fbCase_tests(
	bExecute:= TRUE, 
	bDoorReject:= bDoorReject, 
	stDoorGuardReject:= stCaseRejectReasons_tests.stDoorGuardReject, 
	stProductInstruction:= stProductInstruction_tests, 
	stCodeInfo_Outer:= stCodeInfo_Outer_tests, 
	stCACData:= stCACData_tests, 
	stCACDataHMI:= stCACDataHMI_tests, 
	bDone=> bDone, 
	bBusy=> bBusy, 
	bCACValid=> bCACValid, 
	bCACInvalid=> bCACInvalid, 
	bCheckDuplicates=> bCheckDuplicates, 
	bReadyToValidate=> bReadyToValidate, 
	sRejectCode=> sRejectCode_tests, 
	sCaseContent=> sCaseContent_tests);

bEqualCaseBarcodeCheck := (sTempCaseBarcode = stCACDataHMI_tests.sBarcode);

AssertEquals_BOOL(Expected := TRUE,
                  Actual := bEqualCaseBarcodeCheck,
                  Message := 'HMICaseBarcode not OK on valida data'
);

AssertEquals_STRING(Expected := TO_STRING(sTempCaseBarcode),
                    Actual := TO_STRING(stCACDataHMI_tests.sBarcode),
                    Message := 'HMICaseBarcode String Compare FALSE');
						

TEST_FINISHED();
END_METHOD

METHOD INTERNAL dataHMI02_CaseBarcodeOkOnInalidData
VAR
	fbCase_tests		: FB_CASE_FinaliseData;
	
	bDoorReject			: BOOL;	
	bDone 				: BOOL;
	bBusy				: BOOL;

	bCACValid			: BOOL;
	bCACInvalid			: BOOL;

	bCheckDuplicates	: BOOL;
	bReadyToValidate	: BOOL;
	
	sTempCaseBarcode		: T_CASE_Barcode;
	bEqualCaseBarcodeCheck	: BOOL;			
		
END_VAR

//Data initialization
TestInit(stCACData:= stCACData_tests, stProductInstruction:= stProductInstruction_tests);

//Change some data for test scenario below
stCACData_tests.CaseRejectCode := ''; // data not OK
stCACData_tests.Barcode := 'CaseBarcode';
sTempCaseBarcode := F_CONCAT3(stCACData_tests.Barcode,'(999)','0');
	
TcUnit.TEST('dataHMI02_CaseBarcodeOkOnInalidData');

fbCase_tests(
	bExecute:= TRUE, 
	bDoorReject:= bDoorReject, 
	stDoorGuardReject:= stCaseRejectReasons_tests.stDoorGuardReject, 
	stProductInstruction:= stProductInstruction_tests, 
	stCodeInfo_Outer:= stCodeInfo_Outer_tests, 
	stCACData:= stCACData_tests, 
	stCACDataHMI:= stCACDataHMI_tests, 
	bDone=> bDone, 
	bBusy=> bBusy, 
	bCACValid=> bCACValid, 
	bCACInvalid=> bCACInvalid, 
	bCheckDuplicates=> bCheckDuplicates, 
	bReadyToValidate=> bReadyToValidate, 
	sRejectCode=> sRejectCode_tests, 
	sCaseContent=> sCaseContent_tests);

bEqualCaseBarcodeCheck := (sTempCaseBarcode = stCACDataHMI_tests.sBarcode);

AssertEquals_BOOL(Expected := TRUE,
                  Actual := bEqualCaseBarcodeCheck,
                  Message := 'HMICaseBarcode not OK on valida data'
);

AssertEquals_STRING(Expected := TO_STRING(sTempCaseBarcode),
                    Actual := TO_STRING(stCACDataHMI_tests.sBarcode),
                    Message := 'HMICaseBarcode String Compare FALSE');
						

TEST_FINISHED();
END_METHOD

METHOD INTERNAL dataHMI03_OuterBarcodeOkOnInalidData
VAR
	fbCase_tests		: FB_CASE_FinaliseData;
	
	bDoorReject			: BOOL;	
	bDone 				: BOOL;
	bBusy				: BOOL;

	bCACValid			: BOOL;
	bCACInvalid			: BOOL;

	bCheckDuplicates	: BOOL;
	bReadyToValidate	: BOOL;
	
	sTempCaseBarcode		: T_CASE_Barcode;
	bEqualCaseBarcodeCheck	: BOOL;			
		
END_VAR

//Data initialization
TestInit(stCACData:= stCACData_tests, stProductInstruction:= stProductInstruction_tests);

//Change some data for test scenario below
stCACData_tests.Outer[1].OuterRejectCode := ''; // data not OK
stCACData_tests.Outer[1].Barcode := 'OuterBarcode';
sTempCaseBarcode := F_CONCAT3(stCACData_tests.Outer[1].Barcode,'(999)','0');
	
TcUnit.TEST('dataHMI03_OuterBarcodeOkOnInalidData');

fbCase_tests(
	bExecute:= TRUE, 
	bDoorReject:= bDoorReject, 
	stDoorGuardReject:= stCaseRejectReasons_tests.stDoorGuardReject, 
	stProductInstruction:= stProductInstruction_tests, 
	stCodeInfo_Outer:= stCodeInfo_Outer_tests, 
	stCACData:= stCACData_tests, 
	stCACDataHMI:= stCACDataHMI_tests, 
	bDone=> bDone, 
	bBusy=> bBusy, 
	bCACValid=> bCACValid, 
	bCACInvalid=> bCACInvalid, 
	bCheckDuplicates=> bCheckDuplicates, 
	bReadyToValidate=> bReadyToValidate, 
	sRejectCode=> sRejectCode_tests, 
	sCaseContent=> sCaseContent_tests);

bEqualCaseBarcodeCheck := (sTempCaseBarcode = stCACDataHMI_tests.aOuter[1].sBarcode);

AssertEquals_BOOL(Expected := TRUE,
                  Actual := bEqualCaseBarcodeCheck,
                  Message := 'HMIOuterBarcode not OK on valida data'
);

AssertEquals_STRING(Expected := TO_STRING(sTempCaseBarcode),
                    Actual := TO_STRING(stCACDataHMI_tests.aOuter[1].sBarcode),
                    Message := 'HMIOuterBarcode String Compare FALSE');
						

TEST_FINISHED();
END_METHOD

METHOD INTERNAL dataHMI04_OuterBarcodeNotOkOnValidData
VAR
	fbCase_tests		: FB_CASE_FinaliseData;
	
	bDoorReject			: BOOL;	
	bDone 				: BOOL;
	bBusy				: BOOL;

	bCACValid			: BOOL;
	bCACInvalid			: BOOL;

	bCheckDuplicates	: BOOL;
	bReadyToValidate	: BOOL;
	
	sTempCaseBarcode		: T_CASE_Barcode;
	bEqualCaseBarcodeCheck	: BOOL;			
		
END_VAR

//Data initialization
TestInit(stCACData:= stCACData_tests, stProductInstruction:= stProductInstruction_tests);

//Change some data for test scenario below
stCACData_tests.Outer[1].OuterRejectCode := 'OK'; // data OK
stCACData_tests.Outer[1].Barcode := 'OuterBarcode';
sTempCaseBarcode := F_CONCAT3(stCACData_tests.Outer[1].Barcode,'(999)','1');
	
TcUnit.TEST('dataHMI04_OuterBarcodeNotOkOnValidData');

fbCase_tests(
	bExecute:= TRUE, 
	bDoorReject:= bDoorReject, 
	stDoorGuardReject:= stCaseRejectReasons_tests.stDoorGuardReject, 
	stProductInstruction:= stProductInstruction_tests, 
	stCodeInfo_Outer:= stCodeInfo_Outer_tests, 
	stCACData:= stCACData_tests, 
	stCACDataHMI:= stCACDataHMI_tests, 
	bDone=> bDone, 
	bBusy=> bBusy, 
	bCACValid=> bCACValid, 
	bCACInvalid=> bCACInvalid, 
	bCheckDuplicates=> bCheckDuplicates, 
	bReadyToValidate=> bReadyToValidate, 
	sRejectCode=> sRejectCode_tests, 
	sCaseContent=> sCaseContent_tests);

bEqualCaseBarcodeCheck := (sTempCaseBarcode = stCACDataHMI_tests.aOuter[1].sBarcode);

AssertEquals_BOOL(Expected := TRUE,
                  Actual := bEqualCaseBarcodeCheck,
                  Message := 'HMIOuterBarcode not OK on valida data'
);

AssertEquals_STRING(Expected := TO_STRING(sTempCaseBarcode),
                    Actual := TO_STRING(stCACDataHMI_tests.aOuter[1].sBarcode),
                    Message := 'HMIOuterBarcode String Compare FALSE'
);
						

TEST_FINISHED();
END_METHOD

METHOD INTERNAL dataHMI05_PackBarcodeOkOnInvalidData
VAR
	fbCase_tests		: FB_CASE_FinaliseData;
	
	bDoorReject			: BOOL;	
	bDone 				: BOOL;
	bBusy				: BOOL;

	bCACValid			: BOOL;
	bCACInvalid			: BOOL;

	bCheckDuplicates	: BOOL;
	bReadyToValidate	: BOOL;
	
	sTempCaseBarcode		: T_CASE_Barcode;
	bEqualCaseBarcodeCheck	: BOOL;			
		
END_VAR

//Data initialization
TestInit(stCACData:= stCACData_tests, stProductInstruction:= stProductInstruction_tests);

//Change some data for test scenario below
stCACData_tests.Outer[2].PackRejectCode[4] 	:= ''; // data not OK
stCACData_tests.Outer[2].PackCode[4] 		:= 'PackBarcode';
sTempCaseBarcode := F_CONCAT3(stCACData_tests.Outer[2].PackCode[4],'(999)','0');
	
TcUnit.TEST('dataHMI05_PackBarcodeOkOnInvalidData');

fbCase_tests(
	bExecute:= TRUE, 
	bDoorReject:= bDoorReject, 
	stDoorGuardReject:= stCaseRejectReasons_tests.stDoorGuardReject, 
	stProductInstruction:= stProductInstruction_tests, 
	stCodeInfo_Outer:= stCodeInfo_Outer_tests, 
	stCACData:= stCACData_tests, 
	stCACDataHMI:= stCACDataHMI_tests, 
	bDone=> bDone, 
	bBusy=> bBusy, 
	bCACValid=> bCACValid, 
	bCACInvalid=> bCACInvalid, 
	bCheckDuplicates=> bCheckDuplicates, 
	bReadyToValidate=> bReadyToValidate, 
	sRejectCode=> sRejectCode_tests, 
	sCaseContent=> sCaseContent_tests);

bEqualCaseBarcodeCheck := (sTempCaseBarcode = stCACDataHMI_tests.aOuter[2].aPackCode[4]);

AssertEquals_BOOL(Expected := TRUE,
                  Actual := bEqualCaseBarcodeCheck,
                  Message := 'HMIPackBarcode not OK on valida data'
);

AssertEquals_STRING(Expected := TO_STRING(sTempCaseBarcode),
                    Actual := TO_STRING(stCACDataHMI_tests.aOuter[2].aPackCode[4]),
                    Message := 'HMIPackBarcode String Compare FALSE'
);
						

TEST_FINISHED();
END_METHOD

METHOD INTERNAL dataHMI06_PackBarcodeNotOkOnValidData
VAR
	fbCase_tests		: FB_CASE_FinaliseData;
	
	bDoorReject			: BOOL;	
	bDone 				: BOOL;
	bBusy				: BOOL;

	bCACValid			: BOOL;
	bCACInvalid			: BOOL;

	bCheckDuplicates	: BOOL;
	bReadyToValidate	: BOOL;
	
	sTempCaseBarcode		: T_CASE_Barcode;
	bEqualCaseBarcodeCheck	: BOOL;			
		
END_VAR

//Data initialization
TestInit(stCACData:= stCACData_tests, stProductInstruction:= stProductInstruction_tests);

//Change some data for test scenario below
stCACData_tests.Outer[4].PackRejectCode[10] 	:= 'OK'; // data not OK
stCACData_tests.Outer[4].PackCode[10] 			:= 'PackBarcode';

sTempCaseBarcode := F_CONCAT3(stCACData_tests.Outer[4].PackCode[10],'(999)','1');
	
TcUnit.TEST('dataHMI06_PackBarcodeNotOkOnValidData');

fbCase_tests(
	bExecute:= TRUE, 
	bDoorReject:= bDoorReject, 
	stDoorGuardReject:= stCaseRejectReasons_tests.stDoorGuardReject, 
	stProductInstruction:= stProductInstruction_tests, 
	stCodeInfo_Outer:= stCodeInfo_Outer_tests, 
	stCACData:= stCACData_tests, 
	stCACDataHMI:= stCACDataHMI_tests, 
	bDone=> bDone, 
	bBusy=> bBusy, 
	bCACValid=> bCACValid, 
	bCACInvalid=> bCACInvalid, 
	bCheckDuplicates=> bCheckDuplicates, 
	bReadyToValidate=> bReadyToValidate, 
	sRejectCode=> sRejectCode_tests, 
	sCaseContent=> sCaseContent_tests);

bEqualCaseBarcodeCheck := (sTempCaseBarcode = stCACDataHMI_tests.aOuter[4].aPackCode[10]);

AssertEquals_BOOL(Expected := TRUE,
                  Actual := bEqualCaseBarcodeCheck,
                  Message := 'HMIPackBarcode not OK on valida data'
);

AssertEquals_STRING(Expected := TO_STRING(sTempCaseBarcode),
                    Actual := TO_STRING(stCACDataHMI_tests.aOuter[4].aPackCode[10]),
                    Message := 'HMIPackBarcode String Compare FALSE'
);
						

TEST_FINISHED();
END_METHOD

METHOD INTERNAL main01_FBExecuted_bDoneTRUE
VAR
	fbCase_tests		: FB_CASE_FinaliseData;
	
	bDoorReject			: BOOL;	
	bDone 				: BOOL;
	bBusy				: BOOL;

	bCACValid			: BOOL;
	bCACInvalid			: BOOL;

	bCheckDuplicates	: BOOL;
	bReadyToValidate	: BOOL;
		
END_VAR

//Data initialization
TestInit(stCACData:= stCACData_tests, stProductInstruction:= stProductInstruction_tests);

//Change some data for test scenario below


	
TcUnit.TEST('main01_FBExecuted_bDoneTRUE');

fbCase_tests(
	bExecute:= TRUE, 
	bDoorReject:= bDoorReject, 
	stDoorGuardReject:= stCaseRejectReasons_tests.stDoorGuardReject, 
	stProductInstruction:= stProductInstruction_tests, 
	stCodeInfo_Outer:= stCodeInfo_Outer_tests, 
	stCACData:= stCACData_tests, 
	stCACDataHMI:= stCACDataHMI_tests, 
	bDone=> bDone, 
	bBusy=> bBusy, 
	bCACValid=> bCACValid, 
	bCACInvalid=> bCACInvalid, 
	bCheckDuplicates=> bCheckDuplicates, 
	bReadyToValidate=> bReadyToValidate, 
	sRejectCode=> sRejectCode_tests, 
	sCaseContent=> sCaseContent_tests);



	
AssertEquals_BOOL( Expected	:= TRUE,
			 	   Actual	:= bDone, 
			 	   Message	:= 'FB_CASE_FinaliseData not executed');
						

TEST_FINISHED();
END_METHOD

METHOD INTERNAL main02_bCACValidTrueOnValidData
VAR
	fbCase_tests		: FB_CASE_FinaliseData;
	
	bDoorReject			: BOOL;	
	bDone 				: BOOL;
	bBusy				: BOOL;

	bCACValid			: BOOL;
	bCACInvalid			: BOOL;

	bCheckDuplicates	: BOOL;
	bReadyToValidate	: BOOL;
		
END_VAR

//Data initialization
TestInit(stCACData:= stCACData_tests, stProductInstruction:= stProductInstruction_tests);

//Change some data for test scenario below


	
TcUnit.TEST('main02_bCACValidTrueOnValidData');

fbCase_tests(
	bExecute:= TRUE, 
	bDoorReject:= bDoorReject, 
	stDoorGuardReject:= stCaseRejectReasons_tests.stDoorGuardReject, 
	stProductInstruction:= stProductInstruction_tests, 
	stCodeInfo_Outer:= stCodeInfo_Outer_tests, 
	stCACData:= stCACData_tests, 
	stCACDataHMI:= stCACDataHMI_tests, 
	bDone=> bDone, 
	bBusy=> bBusy, 
	bCACValid=> bCACValid, 
	bCACInvalid=> bCACInvalid, 
	bCheckDuplicates=> bCheckDuplicates, 
	bReadyToValidate=> bReadyToValidate, 
	sRejectCode=> sRejectCode_tests, 
	sCaseContent=> sCaseContent_tests);



	
AssertEquals_BOOL( Expected	:= TRUE,
			 	   Actual	:= bCACValid, 
			 	   Message	:= 'bCACValid wrong value');
						

TEST_FINISHED();
END_METHOD

METHOD INTERNAL main03_bCACInvalidFalseOnValidData
VAR
	fbCase_tests		: FB_CASE_FinaliseData;
	
	bDoorReject			: BOOL;	
	bDone 				: BOOL;
	bBusy				: BOOL;

	bCACValid			: BOOL;
	bCACInvalid			: BOOL;

	bCheckDuplicates	: BOOL;
	bReadyToValidate	: BOOL;
		
END_VAR

//Data initialization
TestInit(stCACData:= stCACData_tests, stProductInstruction:= stProductInstruction_tests);

//Change some data for test scenario below


	
TcUnit.TEST('main03_bCACInvalidFalseOnValidData');

fbCase_tests(
	bExecute:= TRUE, 
	bDoorReject:= bDoorReject, 
	stDoorGuardReject:= stCaseRejectReasons_tests.stDoorGuardReject, 
	stProductInstruction:= stProductInstruction_tests, 
	stCodeInfo_Outer:= stCodeInfo_Outer_tests, 
	stCACData:= stCACData_tests, 
	stCACDataHMI:= stCACDataHMI_tests, 
	bDone=> bDone, 
	bBusy=> bBusy, 
	bCACValid=> bCACValid, 
	bCACInvalid=> bCACInvalid, 
	bCheckDuplicates=> bCheckDuplicates, 
	bReadyToValidate=> bReadyToValidate, 
	sRejectCode=> sRejectCode_tests, 
	sCaseContent=> sCaseContent_tests);



	
AssertEquals_BOOL( Expected	:= FALSE,
			 	   Actual	:= bCACInvalid, 
			 	   Message	:= 'bCACInvalid wrong value');
						

TEST_FINISHED();
END_METHOD

METHOD INTERNAL main04_bCACInvalidTrueOnInvalidData
VAR
	fbCase_tests		: FB_CASE_FinaliseData;
	
	bDoorReject			: BOOL;	
	bDone 				: BOOL;
	bBusy				: BOOL;

	bCACValid			: BOOL;
	bCACInvalid			: BOOL;

	bCheckDuplicates	: BOOL;
	bReadyToValidate	: BOOL;
		
END_VAR

//Data initialization
TestInit(stCACData:= stCACData_tests, stProductInstruction:= stProductInstruction_tests);

//Change some data for test scenario below
stCACData_tests.CaseRejectCode := '';

	
TcUnit.TEST('main04_bCACInvalidTrueOnInvalidData');

fbCase_tests(
	bExecute:= TRUE, 
	bDoorReject:= bDoorReject, 
	stDoorGuardReject:= stCaseRejectReasons_tests.stDoorGuardReject, 
	stProductInstruction:= stProductInstruction_tests, 
	stCodeInfo_Outer:= stCodeInfo_Outer_tests, 
	stCACData:= stCACData_tests, 
	stCACDataHMI:= stCACDataHMI_tests, 
	bDone=> bDone, 
	bBusy=> bBusy, 
	bCACValid=> bCACValid, 
	bCACInvalid=> bCACInvalid, 
	bCheckDuplicates=> bCheckDuplicates, 
	bReadyToValidate=> bReadyToValidate, 
	sRejectCode=> sRejectCode_tests, 
	sCaseContent=> sCaseContent_tests);



	
AssertEquals_BOOL( Expected	:= TRUE,
			 	   Actual	:= bCACInvalid, 
			 	   Message	:= 'bCACInvalid wrong value');
						

TEST_FINISHED();
END_METHOD

METHOD INTERNAL main05_bCACValidFalseOnInvalidData
VAR
	fbCase_tests		: FB_CASE_FinaliseData;
	
	bDoorReject			: BOOL;	
	bDone 				: BOOL;
	bBusy				: BOOL;

	bCACValid			: BOOL;
	bCACInvalid			: BOOL;

	bCheckDuplicates	: BOOL;
	bReadyToValidate	: BOOL;
		
END_VAR

//Data initialization
TestInit(stCACData:= stCACData_tests, stProductInstruction:= stProductInstruction_tests);

//Change some data for test scenario below
stCACData_tests.CaseRejectCode := '';

	
TcUnit.TEST('main05_bCACValidFalseOnInvalidData');

fbCase_tests(
	bExecute:= TRUE, 
	bDoorReject:= bDoorReject, 
	stDoorGuardReject:= stCaseRejectReasons_tests.stDoorGuardReject, 
	stProductInstruction:= stProductInstruction_tests, 
	stCodeInfo_Outer:= stCodeInfo_Outer_tests, 
	stCACData:= stCACData_tests, 
	stCACDataHMI:= stCACDataHMI_tests, 
	bDone=> bDone, 
	bBusy=> bBusy, 
	bCACValid=> bCACValid, 
	bCACInvalid=> bCACInvalid, 
	bCheckDuplicates=> bCheckDuplicates, 
	bReadyToValidate=> bReadyToValidate, 
	sRejectCode=> sRejectCode_tests, 
	sCaseContent=> sCaseContent_tests);



	
AssertEquals_BOOL( Expected	:= FALSE,
			 	   Actual	:= bCACValid, 
			 	   Message	:= 'bCACInvalid wrong value');
						

TEST_FINISHED();
END_METHOD

METHOD INTERNAL main06_FBnotExecuted_bDoneFALSE
VAR
	fbCase_tests		: FB_CASE_FinaliseData;
	
	bDoorReject			: BOOL;	
	bDone 				: BOOL;
	bBusy				: BOOL;

	bCACValid			: BOOL;
	bCACInvalid			: BOOL;

	bCheckDuplicates	: BOOL;
	bReadyToValidate	: BOOL;
		
END_VAR

//Data initialization
TestInit(stCACData:= stCACData_tests, stProductInstruction:= stProductInstruction_tests);

//Change some data for test scenario below


	
TcUnit.TEST('main06_FBnotExecuted_bDoneFALSE');

fbCase_tests(
	bExecute:= FALSE, 
	bDoorReject:= bDoorReject, 
	stDoorGuardReject:= stCaseRejectReasons_tests.stDoorGuardReject, 
	stProductInstruction:= stProductInstruction_tests, 
	stCodeInfo_Outer:= stCodeInfo_Outer_tests, 
	stCACData:= stCACData_tests, 
	stCACDataHMI:= stCACDataHMI_tests, 
	bDone=> bDone, 
	bBusy=> bBusy, 
	bCACValid=> bCACValid, 
	bCACInvalid=> bCACInvalid, 
	bCheckDuplicates=> bCheckDuplicates, 
	bReadyToValidate=> bReadyToValidate, 
	sRejectCode=> sRejectCode_tests, 
	sCaseContent=> sCaseContent_tests);



	
AssertEquals_BOOL( Expected	:= FALSE,
			 	   Actual	:= bDone, 
			 	   Message	:= 'FB_CASE_FinaliseData not executed false');
						

TEST_FINISHED();
END_METHOD

METHOD PUBLIC main07_FBExecuted_bReadyToValidateFALSE
VAR
	fbCase_tests		: FB_CASE_FinaliseData;
	
	bDoorReject			: BOOL;	
	bDone 				: BOOL;
	bBusy				: BOOL;

	bCACValid			: BOOL;
	bCACInvalid			: BOOL;

	bCheckDuplicates	: BOOL;
	bReadyToValidate	: BOOL;
	
		
END_VAR

//Data initialization
TestInit(stCACData:= stCACData_tests, stProductInstruction:= stProductInstruction_tests);

//Change some data for test scenario below


	
TcUnit.TEST('main07_FBExecuted_bReadyToValidateFALSE');

fbCase_tests(
	bExecute:= TRUE, 
	bDoorReject:= bDoorReject, 
	stDoorGuardReject:= stCaseRejectReasons_tests.stDoorGuardReject, 
	stProductInstruction:= stProductInstruction_tests, 
	stCodeInfo_Outer:= stCodeInfo_Outer_tests, 
	stCACData:= stCACData_tests, 
	stCACDataHMI:= stCACDataHMI_tests, 
	bDone=> bDone, 
	bBusy=> bBusy, 
	bCACValid=> bCACValid, 
	bCACInvalid=> bCACInvalid, 
	bCheckDuplicates=> bCheckDuplicates, 
	bReadyToValidate=> bReadyToValidate, 
	sRejectCode=> sRejectCode_tests, 
	sCaseContent=> sCaseContent_tests);



	
AssertEquals_BOOL( Expected	:= TRUE,
			 	   Actual	:= bReadyToValidate, 
			 	   Message	:= 'FB_CASE_FinaliseData executed with bReaduToValidate FALSE');
						

TEST_FINISHED();
END_METHOD

METHOD INTERNAL main08_FBExecuted_bCheckDuplicatesFALSEonOuterDuplicates
VAR
	fbCase_tests		: FB_CASE_FinaliseData;
	
	bDoorReject			: BOOL;	
	bDone 				: BOOL;
	bBusy				: BOOL;

	bCACValid			: BOOL;
	bCACInvalid			: BOOL;

	bCheckDuplicates	: BOOL;
	bReadyToValidate	: BOOL;
		
END_VAR

//Data initialization
TestInit(stCACData:= stCACData_tests, stProductInstruction:= stProductInstruction_tests);

//Change some data for test scenario below
stCACData_tests.Outer[3].Barcode := stCACData_tests.Outer[6].Barcode;

	
TcUnit.TEST('main08_FBExecuted_bCheckDuplicatesFALSEonOuterDuplicates');

fbCase_tests(
	bExecute:= TRUE, 
	bDoorReject:= bDoorReject, 
	stDoorGuardReject:= stCaseRejectReasons_tests.stDoorGuardReject, 
	stProductInstruction:= stProductInstruction_tests, 
	stCodeInfo_Outer:= stCodeInfo_Outer_tests, 
	stCACData:= stCACData_tests, 
	stCACDataHMI:= stCACDataHMI_tests, 
	bDone=> bDone, 
	bBusy=> bBusy, 
	bCACValid=> bCACValid, 
	bCACInvalid=> bCACInvalid, 
	bCheckDuplicates=> bCheckDuplicates, 
	bReadyToValidate=> bReadyToValidate, 
	sRejectCode=> sRejectCode_tests, 
	sCaseContent=> sCaseContent_tests);



	
AssertEquals_BOOL( Expected	:= TRUE,
			 	   Actual	:= bCheckDuplicates, 
			 	   Message	:= 'FB_CASE_FinaliseData executed with bCheckDuplicates FALSE on outer barcode duplicate');
						

TEST_FINISHED();
END_METHOD

METHOD PRIVATE TestInit
VAR_IN_OUT
	stProductInstruction	: ST_PCM_Status;
	stCACData 				: ST_CAC_Data;
END_VAR

VAR	
	rTrigDataInit		: R_TRIG;
	bDataInit			: BOOL;
	iOuter				: INT;
	iPack				: INT;
	sPackNum			: STRING;
	sOuterNum			: STRING;
	sPackCode			: STRING;
END_VAR
	
//MEMSET(ADR(stCACData), 16#00, SIZEOF(stCACData));	

FOR iOuter := 1 TO stProductInstruction.nOutersPerCase DO
	(* Outer number z zerami *)
	sOuterNum := F_StringAddPrefix(INT_TO_STRING(iOuter),2,'0');
	
	(* Write Outers barcodes *)
	stCACData.Outer[iOuter].Barcode    := CONCAT('OUTER', sOuterNum);
	stCACData.Outer[iOuter].OuterCodeStatus := 5;
	stCACData.Outer[iOuter].OuterRejectCode := 'OK';
	
	FOR iPack := 1 TO stProductInstruction.nPacksPerOuter DO
		(* Pack number dwucyfrowy z zerami *)
		sPackNum := F_StringAddPrefix(INT_TO_STRING(iPack),2,'0');			
		(* Sklej pack code *)
		sPackCode := CONCAT(CONCAT('PACK', sPackNum), CONCAT('OUTER', sOuterNum));
		
		(* Write Pack Barcodes / Data*)
		stCACData.Outer[iOuter].PackCode[iPack]			:= sPackCode;
		stCACData.Outer[iOuter].PackCodeStatus[iPack]	:= 5;
		stCACData.Outer[iOuter].PackRejectID[iPack]		:= 0;			
		stCACData.Outer[iOuter].PackRejectCode[iPack]	:= 'OK';
		
					
		stCACData.Outer[iOuter].NumberOfPacks := stProductInstruction.nPacksPerOuter;
		
	END_FOR;
END_FOR;
END_METHOD

END_FUNCTION_BLOCK

// ---- POUs/TcUnit/FB_CASE_DuplicateUpdateToDBTests/FB_CASE_DuplicateUpdateToDBTests.TcPOU
FUNCTION_BLOCK FB_CASE_DuplicateUpdateToDBTests EXTENDS TcUnit.FB_TestSuite

VAR
	
	(* In/Out test 01*)		
	stCACData_01 							: ST_CAC_Data;
	
	stProductInstruction_01		: ST_PCM_Status;
	aOCVPackStatus_01			: ARRAY[1..cMAX_OUTER_STATUS_QUEUE] OF ST_OUTER_Status;	(* Outer status array *)
	aOuterStatus_01				: ARRAY[1..cMAX_OUTER_STATUS_QUEUE] OF ST_OUTER_Status;	(* Outer status array *)
	
	stOCVDataDB_01							: ST_DB_OCVDataCtrl;
	stOACDataDB_01							: ST_DB_OACDataCtrl;
	
	stOuterBarcodeDuplicate_01				: ST_RejectItems;
	stOuterDuplicatedPackCodesFound_01		: ST_RejectItems;
	
	stCodeInfo_Pack_01					: ST_CodeInfo;
	stCodeInfo_Intermediate_01			: ST_CodeInfo;
	stCodeInfo_Outer_01					: ST_CodeInfo;
	
END_VAR

//==============================================================
//MAIN TESTS
//==============================================================

main01_();

METHOD INTERNAL main01_
VAR
	fbCase					: FB_CASE_DuplicateUpdateToDB;
	bIsDuplicateOuter		: BOOL;
	bIsDuplicatePacks		: BOOL;
	

	
END_VAR

//Data initialization
TestInit(stCACData:= stCACData_01, stProductInstruction:= stProductInstruction_01);

//Change some data for test scenario below

	
TcUnit.TEST('main01_');

fbCase(
	bExecute:= TRUE, 
	bUseInterimCodeForValidation:= , 
	aOCVPackStatus:= aOCVPackStatus_01, 
	aOuterStatus:= aOCVPackStatus_01, 
	stOCVDataDB:= stOCVDataDB_01, 
	stOACDataDB:= stOACDataDB_01, 
	stOuterBarcodeDuplicate:=  stOuterBarcodeDuplicate_01, 
	stOuterDuplicatedPackCodesFound:= stOuterDuplicatedPackCodesFound_01, 
	stCodeInfo_Pack:= stCodeInfo_Pack_01, 
	stCodeInfo_Intermediate:= stCodeInfo_Intermediate_01, 
	stCodeInfo_Outer:= stCodeInfo_Outer_01, 
	stCACData:= stCACData_01, 
	bDone=> , 
	bBusy=> , 
	bError=> , 
	nErrorID=> , 
	nOACFilesBlocked=> , 
	nOCVFilesBlocked=> , 
	stDaigOACDataDB=> , 
	stDiagOCVDataDB=> );

	
// AssertEquals_BOOL( Expected	:= ,
// 			 	   Actual	:= , 
// 			 	   Message	:= '');
// 						

TEST_FINISHED();
END_METHOD

METHOD PRIVATE TestInit
VAR_IN_OUT
	stProductInstruction	: ST_PCM_Status;
	stCACData 				: ST_CAC_Data;
END_VAR

VAR	
	rTrigDataInit		: R_TRIG;
	bDataInit			: BOOL;
	iOuter				: INT;
	iPack				: INT;
	sPackNum			: STRING;
	sOuterNum			: STRING;
	sPackCode			: STRING;
END_VAR

stProductInstruction.nOutersPerCase		:= 50;
stProductInstruction.nPacksPerOuter 	:= 10;

stCACData.NumberOfOuters	:= 50;


FOR iOuter := 1 TO stProductInstruction.nOutersPerCase DO
	(* Ustaw outer *)
	stCACData.Outer[iOuter].Barcode    := CONCAT('OUTER', INT_TO_STRING(iOuter));
	stCACData.Outer[iOuter].OuterCodeStatus := 5;
	
	stCACData.Outer[iOuter].OuterRejectID	:= 0;
	
	
	FOR iPack := 1 TO stProductInstruction.nPacksPerOuter DO
		(* Pack number z zerami *)
		sPackNum := CONCAT('0', INT_TO_STRING(iPack));  (* dla 1-9: '01'-'09' *)
		IF iPack = 10 THEN
			sPackNum := '10';
		END_IF;
		
		(* Outer number z zerami dla 1-9 *)
		sOuterNum := CONCAT('0', INT_TO_STRING(iOuter));
		IF iOuter >= 10 THEN
			sOuterNum := INT_TO_STRING(iOuter);
		END_IF;
		
		(* Sklej pack code *)
		sPackCode := CONCAT(CONCAT('PACK', sPackNum), CONCAT('OUTER', sOuterNum));
		
		(* Przypisz *)
		stCACData.Outer[iOuter].PackCode[iPack]			:= sPackCode;
		stCACData.Outer[iOuter].PackCodeStatus[iPack]	:= 5;
		stCACData.Outer[iOuter].PackRejectID[iPack]		:= 0;
		
	END_FOR;
END_FOR;
END_METHOD

END_FUNCTION_BLOCK

// ---- POUs/TcUnit/F_CODE_GetItemAITests/PRG_CODE_GetItemAIManual.TcPOU
PROGRAM PRG_CODE_GetItemAIManual
VAR
	fbCase_DuplicatCheck		: FB_CASE_DuplicatCheck;
	
	(* Init function/method declarations*)
	rTrigDataInit		: R_TRIG;
	bDataInit			: BOOL;
	iOuter				: INT;
	iPack				: INT;
	sPackNum			: STRING;
	sOuterNum			: STRING;
	sPackCode			: STRING;
	
	(* Inputs *)
	bExecute							: BOOL;
	
	(* In/Out *)
	stProductInstruction				: ST_PCM_Status;
	stOuterBarcodeDuplicate				: ST_RejectItems;
	stOuterDuplicatedPackCodesFound		: ST_RejectItems;
	stCaseRejectReasons					: ST_RejectReasonsForCase;
	stRejectReasonForOuters				: ST_RejectReasonsForOuter;	
	stRejectReasonForPacks				: ST_RejectReasonsForPack;	
	
	stCACData 							: ST_CAC_Data;
	
	(* Outputs *)	
	bDone 					: BOOL;
	bBusy					: BOOL;

	bCACValid				: BOOL;
	sRejectCode				: T_MaxString;
	bIsDuplicateOuters		: BOOL;
	bIsDuplicatePacks		: BOOL;
	bReadyToValidate		: BOOL;
	
	stUpdateCACData 		: ST_CAC_Data;
	
	
END_VAR

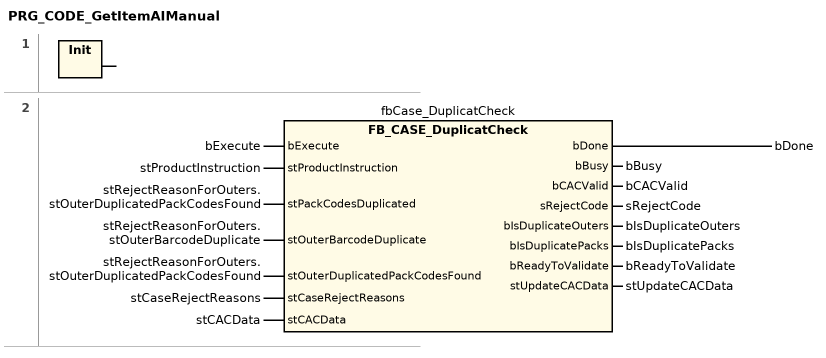
// NETWORK 1
Init();

// NETWORK 2
fbCase_DuplicatCheck(
    bExecute := bExecute,
    stProductInstruction := stProductInstruction,
    stPackCodesDuplicated := stRejectReasonForOuters.stOuterDuplicatedPackCodesFound,
    stOuterBarcodeDuplicate := stRejectReasonForOuters.stOuterBarcodeDuplicate,
    stOuterDuplicatedPackCodesFound := stRejectReasonForOuters.stOuterDuplicatedPackCodesFound,
    stCaseRejectReasons := stCaseRejectReasons,
    stCACData := stCACData,
    bBusy => bBusy,
    bCACValid => bCACValid,
    sRejectCode => sRejectCode,
    bIsDuplicateOuters => bIsDuplicateOuters,
    bIsDuplicatePacks => bIsDuplicatePacks,
    bReadyToValidate => bReadyToValidate,
    stUpdateCACData => stUpdateCACData); // FB_CASE_DuplicatCheck
bDone := fbCase_DuplicatCheck.bDone;

ACTION Init:

rTrigDataInit(CLK := bDataInit);

IF rTrigDataInit.Q THEN
	
stProductInstruction.nOutersPerCase		:= 50;
stProductInstruction.nPacksPerOuter 	:= 10;

	FOR iOuter := 1 TO stProductInstruction.nOutersPerCase DO
		(* Outer number z zerami *)
		sOuterNum := F_StringAddPrefix(INT_TO_STRING(iOuter),2,'0');
		
		(* Write Outers barcodes *)
		stCACData.Outer[iOuter].Barcode    := CONCAT('OUTER', sOuterNum);
		stCACData.Outer[iOuter].OuterCodeStatus := 5;
		
		FOR iPack := 1 TO stProductInstruction.nPacksPerOuter DO
			(* Pack number dwucyfrowy z zerami *)
			sPackNum := F_StringAddPrefix(INT_TO_STRING(iPack),2,'0');			
			(* Sklej pack code *)
			sPackCode := CONCAT(CONCAT('PACK', sPackNum), CONCAT('OUTER', sOuterNum));
			
			(* Write Pack Barcodes *)
			stCACData.Outer[iOuter].PackCode[iPack]			:= sPackCode;
			stCACData.Outer[iOuter].PackCodeStatus[iPack]	:= 5;
			stCACData.Outer[iOuter].PackRejectID[iPack]		:= 0;
			
		END_FOR;
	END_FOR;	
	
END_IF
END_ACTION

END_PROGRAM

// ---- POUs/_Utilites/Addtionals/FB_PulseGenerator_Sync.TcPOU
(* generates one-shot pulses with user-defined period and and sync offset time *)
(* uses GETCPUCOUNTER to synchronise rising edge of timer across multiple FBs *)
FUNCTION_BLOCK FB_PulseGenerator_Sync
VAR_INPUT
	bEnable			: BOOL;		(* set TRUE to enable pulse generation *)
	tPeriod			: TIME;		(* base period for pulse output *)
	nSyncOffset		: DINT;		(* sync offset in ms for rising edge, >0 = phase delay, <0 = phase advance *)
END_VAR
VAR_OUTPUT
	bOutput			: BOOL;		(* one-shot pulse output *)
END_VAR
VAR
	fbCPUCounter	: GETCPUCOUNTER;
	nSystemTime64	: T_ULARGE_INTEGER;
	nSystemTime		: UDINT;
	nLastSystemTime	: UDINT;
END_VAR
(*
-------------------------------------------------------------------------------------------------
Date		Version	Author	Comments
-------------------------------------------------------------------------------------------------
30/01/2015	3.00.00	PB		Initial release

-------------------------------------------------------------------------------------------------
*)

(* enabled and tBaseTime is specified *)
IF bEnable = TRUE AND tPeriod > T#0ms THEN

	(* load global CPU counter value into 64-bit nSystemTime *)
	fbCPUCounter(
		cpuCntLoDW	=> nSystemTime64.dwLowPart,
		cpuCntHiDW	=> nSystemTime64.dwHighPart
	);

	(* phase delay *)
	IF nSyncOffset > 0 THEN

		(* subtract nTimeOffset from system timer *)
		nSystemTime64 := UInt64Sub64(nSystemTime64, UInt32x32To64(ABS(nSyncOffset), 10000));

	(* phase advance *)
	ELSIF nSyncOffset < 0 THEN

		(* add nTimeOffset from system timer *)
		nSystemTime64 := UInt64Add64(nSystemTime64, UInt32x32To64(ABS(nSyncOffset), 10000));
	END_IF

	(* convert nSystemTime from 1= 100ns to 1 = 1ms *)
	nSystemTime64 := UInt64Div64(nSystemTime64, UInt32x32To64(10000, 1));

	(* nSystemTime is sawtooth wave from 0 to tPeriod in ms *)
	nSystemTime := nSystemTime64.dwLowPart MOD TIME_TO_UDINT(tPeriod);

	(* nSystemTime has re-started, convert nLastSystemTime to tPeriod *)
	IF nSystemTime < nLastSystemTime MOD TIME_TO_UDINT(tPeriod) THEN

		bOutput := TRUE;

	(* nSystemTime >= nLastSystemTime *)
	ELSE

		bOutput := FALSE;
	END_IF

	(* store last system time *)
	nLastSystemTime := nSystemTime;

(* disabled or tBaseTime = 0ms *)
ELSE

	bOutput := FALSE;
END_IF

END_FUNCTION_BLOCK

// ---- POUs/_Utilites/Addtionals/PRG_ButtonsHandler.TcPOU
PROGRAM PRG_ButtonsHandler
VAR
	rTrig			: R_TRIG;
	tTimer			: TOF;
	tTriggerTime	: TIME := T#100MS;
	bTimerOn		: BOOL;
END_VAR


rTrig(CLK:= GVL.bSiemensTriggerButton);

tTimer(IN:= bTimerOn, PT:= tTriggerTime);

IF rTrig.Q THEN
	bTimerOn := TRUE;	
ELSIF tTimer.ET = T#0S THEN
	bTimerOn := FALSE;
END_IF

GVL.bSiemensTriggerOutput := tTimer.Q;

END_PROGRAM

// ---- POUs/_Utilites/CAMERAS/FB_SCANNER_HikrobotEXT.TcPOU
FUNCTION_BLOCK FB_SCANNER_HikrobotEXT
VAR_INPUT
	bEnableReceive					: BOOL;
	bEnableSend						: BOOL;
	strScannerIPAddr				: T_IPv4Addr	:= '192.168.1.45';
	nReceiveScannerPortNo			: UINT			:= 2010;
	nSendScannerPortNo				: UINT			:= 4001;	
	stRequestCommand				: E_TCPIP_RequescCommand; (* tutaj powinna byc strukruta z eRequestCommand plus parametry: 0,1 etc *)
	bSendCommand					: BOOL;
	bExecutedCommandSend			: BOOL;
END_VAR

VAR_OUTPUT
	eSocketReceiveState		: E_SocketConnectionState;
	eSocketSendState		: E_SocketConnectionState;
END_VAR

VAR
	fbTCPPortCtrl_Receive	: FB_TCP_ClientPortCtrl;
	bReceiveConnected		: BOOL;
	fbTCPortCtrl_Send		: FB_TCP_ClientPortCtrl;
	bSendConnected			: BOOL;
	fbTCPReceive			: FB_ReceiveString;
	bReceiveExpected		: BOOL;
	fbTCPReceiveAfterSend	: FB_ReceiveString;	
	strTCPRxStringReply		: T_MaxString;
	strTCPRxString			: T_MaxString;
	strTCPRxString_Reply	: T_MaxString;
	ftrigEnable				: F_TRIG;
	bReInitialiseTCP		: BOOL;
	fbTON_TcpTimeout		: TON;
	
	nIndex					: UINT;
	nIndexReply				: UINT;
	nIndex2					: UINT;
	
	/////// send command
	
	fbTCPSend				: FB_SocketSend;
	rTrigSend				: R_TRIG;
	rTrigDataReceived		: R_TRIG;
	rTrigSendCommand		: R_TRIG;
	nCommandNo				: UINT := 1;
	fTrigTCPSendDone		: F_TRIG;
	nSendErrId				: UDINT;
	strTCPCommand			: STRING(20);
	strReplyString			: STRING(20);
	strTCPLastCommand		: STRING(20);
	strLastReplyString		: STRING(20);
	bReplyOK				: BOOL;
	tHeartbeatInterval		: TIME := T#5S;
	eRequestCommand			: E_TCPIP_RequescCommand;
	
	(* SEND SEQUENCE VARIABLE *)
	
	eSendSequenceSTATE		: E_TCPIP_SEND_STATE;
	bSendRequest			: BOOL;
	rTrigSendRequest		: R_TRIG;
END_VAR


Connect();

Receive();

//Send();

Send_Sequence();

ACTION Connect:

(* TCP Receive Socket establish connect *)
fbTCPPortCtrl_Receive(
	bEnable				:= bEnableReceive, 
	strRemoteIPAddr		:= strScannerIPAddr, 
	nRemotePortNo		:= nReceiveScannerPortNo, 
	tReconnectTime		:= T#20S, 
	eSocketState		=> eSocketReceiveState, 
	bError				=> , 
	nErrorID			=>,
	bConnected			=> bReceiveConnected
 );
	
(* TCP Send Socket establish connect *)
fbTCPortCtrl_Send(
	bEnable				:= bEnableSend, 
	strRemoteIPAddr		:= strScannerIPAddr, 
	nRemotePortNo		:= nSendScannerPortNo, 
	tReconnectTime		:= T#20S, 
	eSocketState		=> eSocketSendState, 
	bError				=> , 
	nErrorID			=>, 
	bConnected			=> bSendConnected
);
END_ACTION

ACTION Receive:

ftrigEnable(CLK := bEnableReceive);
IF ftrigEnable.Q THEN
	strTCPRxString := ''; (* clears input buffer *)
END_IF

(* poll TCP port receive string *)
fbTCPReceive(
	bEnable			:= fbTCPPortCtrl_Receive.bConnected,
	hSocket			:= fbTCPPortCtrl_Receive.hSocket,
	tUpdateTime		:= T#100MS,
	strTCPRxString	:= strTCPRxString
);


//*************** quick patch ****************//
IF fbTCPReceive.bDataReceived THEN
	GVL.aTCPxStrings[nIndex] := strTCPRxString;
	nIndex := nIndex + 1;
	strTCPRxString := '';
END_IF
	
IF nIndex = 20 THEN
	nIndex := 0;
	FOR nIndex2 := 0 TO 20 DO
		GVL.aTCPxStrings[nIndex2] := '';		
	END_FOR
END_IF

IF nIndexReply = 20 THEN
	nIndexReply := 0;
	FOR nIndex2 := 0 TO 20 DO
		GVL.aTCPxStringsReply[nIndex2] := '';		
	END_FOR
END_IF

//*************** quick patch ****************//
END_ACTION

ACTION Send:

rTrigSend(CLK := bSendCommand);
IF rTrigSend.Q THEN
	strTCPCommand 	:= GVL.aHikrobotCtrlCommands[nCommandNo];	
END_IF

fbTCPSend(
	sSrvNetId	:= '',
	hSocket		:= fbTCPortCtrl_Send.hSocket,
	cbLen		:= TO_UDINT(LEN(strTCPCommand)),
	pSrc		:= ADR(strTCPCommand),
	bExecute	:= rTrigSend.Q,
	tTimeout	:= T#1s
);

(* send data complete *)
fTrigTCPSendDone(CLK := fbTCPSend.bBusy);
(* TCP send complete *)

IF fbTCPSend.bError = TRUE THEN
	nSendErrId := fbTCPSend.nErrId;
ELSE
	nSendErrId := 0;	
END_IF

IF fTrigTCPSendDone.Q = TRUE THEN

	(* clear strTCPCommand *)
	strTCPCommand := '';

	(* close off fbSendTCPData *)
	fbTCPSend(bExecute := FALSE);
END_IF


// expece response after sending command
fbTCPReceiveAfterSend(
	bEnable			:= bSendCommand AND fbTCPortCtrl_Send.bConnected,
	hSocket			:= fbTCPortCtrl_Send.hSocket,
	tUpdateTime		:= T#100MS,
	strTCPRxString	:= strTCPRxString_Reply
);
END_ACTION

ACTION Send_Sequence:

rTrigSendCommand(CLK := bSendCommand);

IF rTrigSendCommand.Q  THEN	
	IF stRequestCommand <> 0 THEN
		eRequestCommand	:= stRequestCommand;
	END_IF	
END_IF

fbTCPSend(
	sSrvNetId	:= '',
	hSocket		:= fbTCPortCtrl_Send.hSocket,
	cbLen		:= TO_UDINT(LEN(strTCPCommand)),
	pSrc		:= ADR(strTCPCommand),
	bExecute	:= fbTCPSend.cbLen > 0 AND fbTCPSend.bBusy = FALSE,
	tTimeout	:= T#1S
);
	
	(* send data complete *)
fTrigTCPSendDone(CLK := fbTCPSend.bBusy);
IF fTrigTCPSendDone.Q = TRUE THEN

	IF fbTCPSend.bError = TRUE THEN
		bReInitialiseTCP := TRUE;
	END_IF

	strTCPLastCommand 	:= strTCPCommand;
	strLastReplyString	:= strReplyString;
	eRequestCommand 	:= E_TCPIP_RequescCommand.NONE;
	(* close off fbSendTCP *)
	fbTCPSend(bExecute 	:= FALSE);
	
	(* expece to receive reply after send finished *)
	bReceiveExpected	:= TRUE;
	
END_IF

fbTCPReceiveAfterSend(
	bEnable			:= fbTCPortCtrl_Send.bConnected,
	hSocket			:= fbTCPortCtrl_Send.hSocket,
	tUpdateTime		:= T#100MS,
	strTCPRxString	:= strTCPRxStringReply
);

rTrigDataReceived(CLK:=fbTCPReceiveAfterSend.bDataReceived);
IF rTrigDataReceived.Q THEN
	(*  veryfi valide response *)
	
	IF strLastReplyString = strTCPRxStringReply THEN
		bReplyOK := TRUE;
	ELSE		
		bReplyOK := FALSE;			
	END_IF
	
	GVL.aTCPxStringsReply[nIndexreply] 	:= strTCPRxStringReply;
	nIndexReply	 						:= nIndexReply + 1;
	strTCPRxStringReply 				:= '';
	bReceiveExpected					:= FALSE;
	
END_IF

// HeartBeat send every tHeartbeatInterval, if heartbead doesent reply do bReInitialiseTCP := TRUE
fbTON_TcpTimeout(
	IN	:= fbTCPortCtrl_Send.bConnected,
 	PT	:= tHeartbeatInterval
);
IF fbTON_TcpTimeout.Q AND (eRequestCommand = E_TCPIP_RequescCommand.NONE) THEN
	eRequestCommand 	:= E_TCPIP_RequescCommand.HeartbeatCheck;	
	fbTON_TcpTimeout(IN := FALSE);
END_IF
//////////////////////////// heartbeat handeling end ///////////////////////////////////////////////

CASE eRequestCommand OF
	
	E_TCPIP_RequescCommand.NONE:		
		strTCPCommand 	:= '';	
		strReplyString	:= '';		
	
	E_TCPIP_RequescCommand.GetUserCur:		
		strTCPCommand 	:= '<Get,UserCur>';	
		strReplyString	:= '<Get,UserCur,6>';	
		
	E_TCPIP_RequescCommand.WrongReply:		
		strTCPCommand 	:= '<Get,UserCur>';	
		strReplyString	:= '<Get,UserCur,2>';
	
	E_TCPIP_RequescCommand.HeartbeatCheck:		
		strTCPCommand 	:= '<Get,RunMode>';	
		strReplyString	:= '<Get,RunMode,0>';		
		
	E_TCPIP_RequescCommand.SetAquisitonModeON:
		strTCPCommand 	:= '<Set,Acq,1>';	
		strReplyString	:= '<Set,Acq,OK>';	
		
	E_TCPIP_RequescCommand.SetAquisitionModeOFF:
		strTCPCommand 	:= '<Set,Acq,0>';	
		strReplyString	:= '<Set,Acq,OK>';
	
END_CASE
END_ACTION

END_FUNCTION_BLOCK

// ---- POUs/_Utilites/TCP_FB/FB_TCP_ClientPortCtrl.TcPOU
FUNCTION_BLOCK FB_TCP_ClientPortCtrl

VAR_INPUT
	bEnable				: BOOL;			(* set TRUE to enable TCP connection *)
	strRemoteIPAddr		: T_IPv4Addr;	(* IP address for remote device *)
	nRemotePortNo		: UINT;			(* port number for remote device *)	
	tReconnectTime		: TIME:= DEFAULT_ADS_TIMEOUT;
END_VAR

VAR_OUTPUT	
	eSocketState		: E_SocketConnectionState;
	hSocket				: T_HSOCKET;
	bError				: BOOL;
	nErrorID			: UDINT;
	bConnected			: BOOL;
END_VAR

VAR	
	fbTCPSocketCtrl		: FB_ClientServerConnection;
	eTCPState			: E_TCPIP_StateWP;
	strTargetIPAddr		: T_IPv4Addr;
	nTargetPortNo		: UDINT;
END_VAR

CASE eTCPState OF
	
	E_TCPIP_StateWP.E_TCPIP_IDLE:
	
		IF bEnable THEN			
			strTargetIPAddr	:= strRemoteIPAddr;
			nTargetPortNo	:= nRemotePortNo;
		
			eTCPState		:= E_TCPIP_StateWP.E_TCPIP_CONNECT;	
		END_IF
	
	E_TCPIP_StateWP.E_TCPIP_CONNECT:
	
		IF NOT bEnable OR fbTCPSocketCtrl.bError  THEN
			eTCPState:= E_TCPIP_StateWP.E_TCPIP_DISCONNECT;
		END_IF
	
	(* close TCP connection *)
	E_TCPIP_StateWP.E_TCPIP_DISCONNECT:

		(* TCP port has been closed, fbTCPSocketCtrl.bEnable FALSE in this state *)
		IF eSocketState = eSOCKET_DISCONNECTED THEN
			eTCPState := E_TCPIP_StateWP.E_TCPIP_IDLE;
		END_IF
		
	(* unknown state *)
ELSE

	eTCPState := E_TCPIP_StateWP.E_TCPIP_IDLE;

END_CASE


(* TCP port connection ctrl *)
fbTCPSocketCtrl(
	sSrvNetID	:= '',
	nMode		:= LISTEN_MODE_CLOSEALL, (*LISTEN_MODE_USEOPENED, CONNECT_MODE_ENABLEDBG, LISTEN_MODE_CLOSEALL*)
	sRemoteHost	:= strTargetIPAddr,
	nRemotePort	:= nTargetPortNo,
	bEnable		:= eTCPState = E_TCPIP_StateWP.E_TCPIP_CONNECT,
	tReconnect	:= tReconnectTime,
	bError		=> bError,
	nErrID		=> ,
	hSocket		=> hSocket,  
	eState		=> eSocketState
);

IF NOT fbTCPSocketCtrl.bBusy THEN
	nErrorID:= fbTCPSocketCtrl.nErrId;
END_IF

bConnected:= eSocketState = eSOCKET_CONNECTED;

END_FUNCTION_BLOCK

// ---- POUs/_Utilites/TCP_FB/FB_ReceiveString.TcPOU
FUNCTION_BLOCK FB_ReceiveString

VAR_INPUT
	bEnable				: BOOL;			(* set TRUE to enable periodic TCP data receive *)
	hSocket				: T_HSocket;	(* TCP socket *)
	tUpdateTime			: TIME;			(* receive update rate *)
	nSyncOffset			: DINT;			(* ms offset to spread TCP Server access loading *)
END_VAR

VAR_IN_OUT
	strTCPRxString		: T_MaxString;	(* string to which incoming TCP data will be appended *)
END_VAR

VAR_OUTPUT
	bDone				: BOOL;			(* TRUE = complete *)
	bBusy				: BOOL;			(* TRUE = in progress *)
	bError 				: BOOL;			(* TRUE = error *)
	nErrorID			: UDINT;		(* error code *)
	bDataReceived		: BOOL;			(* TRUE = data received *)
END_VAR

VAR
	fbTCPReceive		: FB_SocketReceive;
	strTCPRxChars		: T_MaxString;
	bTCPReceive			: BOOL:= FALSE;
	fbTimer				: FB_PulseGenerator_Sync;
	nMaxBytes			: UDINT;
END_VAR


(* TCP update timer *)
fbTimer(
	bEnable		:= bEnable,
	tPeriod		:= tUpdateTime,
	nSyncOffset	:= nSyncOffset
);

(* TCP update timer elapsed and fbTCPReceive is not active *)
IF fbTimer.bOutput = TRUE THEN

	(* max number of bytes that can be received into strTCPRxString on next cycle *)
	nMaxBytes := SIZEOF(strTCPRxString) - LEN2(ADR(strTCPRxString)) - 1;

	(* clear strTCPRxChars *)
	MEMSET(ADR(strTCPRxChars), 16#00, SIZEOF(strTCPRxChars));

	(* strTCPRxString has space for 1 or more bytes *)
	IF nMaxBytes > 0 THEN

		(* receive data from TCP port *)
		bTCPReceive := TRUE;
		bBusy := TRUE;
	END_IF

	(* clear outputs *)
	bDone := FALSE;
	bError := FALSE;
	nErrorID := 0;
	bDataReceived := FALSE;

(* TPC receive not active *)
ELSIF bTCPReceive = FALSE THEN

	(* clear outputs *)
	bDone := FALSE;
	bBusy := FALSE;
	bError := FALSE;
	nErrorID := 0;
	
	bDataReceived := FALSE;
END_IF

fbTCPReceive(
	sSrvNetId	:= , 
	hSocket		:= hSocket, 
	cbLen		:= nMaxBytes, 
	pDest		:= ADR(strTCPRxChars), 
	bExecute	:= bTCPReceive, 
	tTimeout	:= T#500MS, 
	bBusy		=> bBusy
);
	
	
(* receive TCP data complete *)
IF bTCPReceive = TRUE AND fbTCPReceive.bBusy = FALSE THEN

	(* receive TCP data completed OK *)
	IF fbTCPReceive.bError = FALSE THEN

		(* data bytes received *)
		IF fbTCPReceive.nRecBytes > 0 THEN

			(* append returned data to TCP data string *)
			strTCPRxString := CONCAT(strTCPRxString, strTCPRxChars); //CONCAT limited to return String(255)
			bDataReceived := TRUE;
		END_IF

		(* clear errors flags if currently no error*)
		bError := FALSE;
		nErrorID := 0;
	(* receive data error *)
	ELSE

		bDataReceived := FALSE;
		bError := TRUE;
		nErrorID := fbTCPReceive.nErrId;
		bDone := FALSE;
	END_IF

	(* clear TCP Receive flag *)
	bTCPReceive := FALSE;

	(* update outputs *)
	bDone := TRUE;
	bBusy := FALSE;

	(* close off fbReceiveTCPData *)
	fbTCPReceive(bExecute := FALSE);
END_IF

END_FUNCTION_BLOCK

// ---- POUs/_Utilites/CAMERAS/F_CREATE_MESSAGE.TcPOU
FUNCTION F_CREATE_MESSAGE : BOOL
VAR_INPUT
END_VAR
VAR
END_VAR

END_FUNCTION

// ---- POUs/_Utilites/METS/Common LIB/08_SOFTWARE LIB/AI Codes And Validation FBs/FB_CODE_ClearCodeInfo.TcPOU
FUNCTION_BLOCK FB_CODE_ClearCodeInfo
VAR_INPUT
END_VAR
VAR_IN_OUT
	stCodeInfo						: ST_CodeInfo;
END_VAR
VAR
	sMemoUserField1					: STRING;
	sMemoUserField2					: STRING;
	sMemoUserField3					: STRING;
END_VAR

IF stCodeInfo.stGTIN.nListPosition = 0 THEN
	MEMSET(ADR(stCodeInfo.stGTIN), 16#00, SIZEOF(stCodeInfo.stGTIN));
	stCodeInfo.stGTIN.sFieldName :='GTIN';
	stCodeInfo.stGTIN.nGS1_AI := 1;
END_IF
IF stCodeInfo.stBatchID.nListPosition  = 0 THEN
	MEMSET(ADR(stCodeInfo.stBatchID), 16#00, SIZEOF(stCodeInfo.stBatchID));
	stCodeInfo.stBatchID.sFieldName :='BatchID';
	stCodeInfo.stBatchID.nGS1_AI := 10;
END_IF
IF stCodeInfo.stSerialCode.nListPosition = 0 THEN
	MEMSET(ADR(stCodeInfo.stSerialCode), 16#00, SIZEOF(stCodeInfo.stSerialCode));
	stCodeInfo.stSerialCode.sFieldName :='SerialCode';
	stCodeInfo.stSerialCode.nGS1_AI := 21;
END_IF
IF stCodeInfo.stProductionOrder.nListPosition  = 0 THEN
	MEMSET(ADR(stCodeInfo.stProductionOrder), 16#00, SIZEOF(stCodeInfo.stProductionOrder));
	stCodeInfo.stProductionOrder.sFieldName :='ProductionOrder';
	stCodeInfo.stProductionOrder.nGS1_AI := 91;
END_IF
IF stCodeInfo.stCryptoCode.nListPosition = 0 THEN
	MEMSET(ADR(stCodeInfo.stCryptoCode), 16#00, SIZEOF(stCodeInfo.stCryptoCode));
	stCodeInfo.stCryptoCode.sFieldName :='CryptoCode';
	stCodeInfo.stCryptoCode.nGS1_AI := 93;
END_IF
IF stCodeInfo.stRSKU.nListPosition = 0 THEN
	MEMSET(ADR(stCodeInfo.stRSKU), 16#00, SIZEOF(stCodeInfo.stRSKU));
	stCodeInfo.stRSKU.sFieldName :='SKU';
	stCodeInfo.stRSKU.nGS1_AI := 240;
END_IF
IF stCodeInfo.stMRP.nListPosition = 0 THEN
	MEMSET(ADR(stCodeInfo.stMRP), 16#00, SIZEOF(stCodeInfo.stMRP));
	stCodeInfo.stMRP.sFieldName :='MRP';
	stCodeInfo.stMRP.nGS1_AI := 8005;
END_IF
IF stCodeInfo.stBrandSpecification.nListPosition = 0 THEN
	MEMSET(ADR(stCodeInfo.stBrandSpecification), 16#00, SIZEOF(stCodeInfo.stBrandSpecification));
	stCodeInfo.stBrandSpecification.sFieldName := 'BrandSpec';
	stCodeInfo.stBrandSpecification.nGS1_AI := 92;
END_IF
IF stCodeInfo.stProduceDate.nListPosition = 0 THEN
	MEMSET(ADR(stCodeInfo.stProduceDate), 16#00, SIZEOF(stCodeInfo.stProduceDate));
	stCodeInfo.stProduceDate.sFieldName :='ProduceDate';
	stCodeInfo.stProduceDate.nGS1_AI := 94;
END_IF
IF stCodeInfo.stUserField3.nListPosition  = 0THEN
	sMemoUserField3 := stCodeInfo.stUserField3.sFieldName;
	MEMSET(ADR(stCodeInfo.stUserField3), 16#00, SIZEOF(stCodeInfo.stUserField3));
	stCodeInfo.stUserField3.sFieldName :=sMemoUserField3;
	stCodeInfo.stUserField3.nGS1_AI := 95;
END_IF

END_FUNCTION_BLOCK

// ---- POUs/_Utilites/METS/Common LIB/08_SOFTWARE LIB/AI GS1 Codes And Validation FBs/FB_GS1_ClearCodeInfo.TcPOU
FUNCTION_BLOCK FB_GS1_ClearCodeInfo
VAR_INPUT
END_VAR
VAR_IN_OUT
	stCodeInfo						: ST_GS1_CodeInfo;
END_VAR
VAR
	nItemIndex		: INT ;
END_VAR

FOR nItemIndex :=1 TO cMAX_VALIDATION_ITEMS DO
	IF stCodeInfo.stGS1_Field[nItemIndex].eGS1_AIType = GS1_00   THEN
		MEMSET(ADR(stCodeInfo.stGS1_Field[nItemIndex]), 16#00, SIZEOF(stCodeInfo.stGS1_Field[nItemIndex]));
		stCodeInfo.stGS1_Field[nItemIndex].sFieldName :='Field Undefined';
	END_IF
END_FOR

END_FUNCTION_BLOCK

// ---- POUs/_Utilites/METS/Common LIB/08_SOFTWARE LIB/AI GS1 Codes And Validation FBs/FB_GS1_ValidateExplicitCode.TcPOU
 FUNCTION_BLOCK FB_GS1_ValidateExplicitCode
VAR_INPUT
	sFullCode					: T_MaxString;
	stCodeInfo				: ST_GS1_CodeInfo;
	stGS1_AI_Definition			: ST_GS1_AI_Definition;
END_VAR
VAR_OUTPUT
	bValidationOK				: BOOL;
	bEntireCodeLengthOK		: BOOL;

	(*bGS1_01_OK	: BOOL;
	bGS1_10_OK	: BOOL;
	bGS1_11_OK	: BOOL;
	bGS1_15_OK	: BOOL;
	bGS1_17_OK	: BOOL;
	bGS1_21_OK	: BOOL;
	bGS1_91_OK	: BOOL;
	bGS1_92_OK	: BOOL;
	bGS1_93_OK	: BOOL;
	bGS1_94_OK	: BOOL;
	bGS1_240_OK	: BOOL;
	bGS1_8005_OK	: BOOL;

	(*Fixed string lenght according to max string lenght form GS1*)
	sGS1_01		:STRING(14);
	sGS1_10		:STRING(20);
	sGS1_11		:STRING(6);
	sGS1_15		:STRING(6);
	sGS1_17		:STRING(6);
	sGS1_21		:STRING(21);
	sGS1_91		:STRING(90);
	sGS1_92		:STRING(90);
	sGS1_93		:STRING(90);
	sGS1_94		:STRING(90);
	sGS1_240		:STRING(30);
	sGS1_8005	:STRING(6);*)

END_VAR
VAR
	stItem			: ST_GS1_CodeValidation;
	nItemIndex		: INT;

	sAI_01ToValidateAgainst		: STRING(14);

	bGS1_01_OK	: BOOL;
	bGS1_10_OK	: BOOL;
	bGS1_11_OK	: BOOL;
	bGS1_15_OK	: BOOL;
	bGS1_17_OK	: BOOL;
	bGS1_21_OK	: BOOL;
	bGS1_240_OK	: BOOL;
	bGS1_8005_OK	: BOOL;
	bGS1_8006_OK	: BOOL;
	bGS1_8008_OK	: BOOL;
	bGS1_91_OK	: BOOL;
	bGS1_92_OK	: BOOL;
	bGS1_93_OK	: BOOL;
	bGS1_94_OK	: BOOL;

	bNON_GS1_01_OK	: BOOL;
	bNON_GS1_02_OK	: BOOL;
	bNON_GS1_03_OK	: BOOL;
	bNON_GS1_04_OK	: BOOL;
	bNON_GS1_05_OK	: BOOL;
	bNON_GS1_06_OK	: BOOL;
	bNON_GS1_07_OK	: BOOL;
	bNON_GS1_08_OK	: BOOL;
	bNON_GS1_09_OK	: BOOL;
	bNON_GS1_10_OK	: BOOL;

	(*Fixed string lenght according to max string lenght form GS1*)
	sGS1_01		:STRING(14);
	sGS1_10		:STRING(20);
	sGS1_11		:STRING(6);
	sGS1_15		:STRING(6);
	sGS1_17		:STRING(6);
	sGS1_21		:STRING(20);
	sGS1_240		:STRING(30);
	sGS1_8005	:STRING(6);
	sGS1_8006	:STRING(18);
	sGS1_8008	:STRING(12);
	sGS1_91		:STRING(90);
	sGS1_92		:STRING(90);
	sGS1_93		:STRING(90);
	sGS1_94		:STRING(90);

	sNON_GS1_01		:STRING(255);
	sNON_GS1_02		:STRING(255);
	sNON_GS1_03		:STRING(255);
	sNON_GS1_04		:STRING(255);
	sNON_GS1_05		:STRING(255);
	sNON_GS1_06		:STRING(255);
	sNON_GS1_07		:STRING(255);
	sNON_GS1_08		:STRING(255);
	sNON_GS1_09		:STRING(255);
	sNON_GS1_10		:STRING(255);

END_VAR

IF	stCodeInfo.nEntireLength = 0 THEN
	bEntireCodeLengthOK := FALSE;
	RETURN;
ELSIF	stCodeInfo.nEntireLength = stCodeInfo.nMinLength THEN
	bEntireCodeLengthOK := (LEN(sFullCode) = stCodeInfo.nEntireLength) OR NOT stCodeInfo.bValidateEntireLength;
ELSE
	bEntireCodeLengthOK := (LEN(sFullCode) >= stCodeInfo.nMinLength  AND   LEN(sFullCode) <= stCodeInfo.nEntireLength) OR NOT stCodeInfo.bValidateEntireLength;
END_IF

CASE stCodeInfo.eCodeLvlType OF

	E_LEVEL1:
		sAI_01ToValidateAgainst := stGS1_AI_Definition.stAI_01_Lvl1.sDataField;
	E_LEVEL2:
		sAI_01ToValidateAgainst := stGS1_AI_Definition.stAI_01_Lvl2.sDataField;
	E_LEVEL3:
		sAI_01ToValidateAgainst := stGS1_AI_Definition.stAI_01_Lvl3.sDataField;
ELSE
		sAI_01ToValidateAgainst := '';
END_CASE

sGS1_01		:='';
sGS1_10		:='';
sGS1_11		:='';
sGS1_15		:='';
sGS1_17		:='';
sGS1_21		:='';
sGS1_91		:='';
sGS1_92		:='';
sGS1_93		:='';
sGS1_94		:='';
sGS1_240		:='';
sGS1_8005	:='';

(*********************** GS1_01**************************************)
bGS1_01_OK := FALSE;
sGS1_01 := F_GS1_GetItem(sFullCode, GS1_01, stCodeInfo);

FOR nItemIndex :=1 TO cMAX_VALIDATION_ITEMS DO
	IF stCodeInfo.stGS1_Field[nItemIndex].eGS1_AIType =  GS1_01 THEN
		stItem := stCodeInfo.stGS1_Field[nItemIndex];
		IF stItem.bValidate THEN
			IF (LEN(sGS1_01) =  stItem.nCodeLength OR stItem.nCodeLength = 0)  AND  (sGS1_01 = sAI_01ToValidateAgainst OR sAI_01ToValidateAgainst = '') THEN
				bGS1_01_OK := TRUE;
			END_IF
		ELSE
			bGS1_01_OK := TRUE;
		END_IF
		EXIT;
	END_IF
END_FOR

(*********************** ********************************************)
(*********************** GS1_10**************************************)
bGS1_10_OK := FALSE;
sGS1_10 := F_GS1_GetItem(sFullCode, GS1_10, stCodeInfo);

FOR nItemIndex :=1 TO cMAX_VALIDATION_ITEMS DO
	IF stCodeInfo.stGS1_Field[nItemIndex].eGS1_AIType =  GS1_10 THEN
		stItem := stCodeInfo.stGS1_Field[nItemIndex];
		IF stItem.bValidate THEN
			IF (LEN(sGS1_10) = stItem.nCodeLength OR stItem.nCodeLength = 0) AND ( sGS1_10 =  stGS1_AI_Definition.stAI_10.sDataField OR stGS1_AI_Definition.stAI_10.sDataField = '') THEN
				bGS1_10_OK := TRUE;
			END_IF
		ELSE
			bGS1_10_OK := TRUE;
		END_IF
		EXIT;
	END_IF
END_FOR

(*********************** ********************************************)
(*********************** GS1_11**************************************)
bGS1_11_OK := FALSE;
sGS1_11 := F_GS1_GetItem(sFullCode, GS1_11, stCodeInfo);

FOR nItemIndex :=1 TO cMAX_VALIDATION_ITEMS DO
	IF stCodeInfo.stGS1_Field[nItemIndex].eGS1_AIType =  GS1_11 THEN
		stItem := stCodeInfo.stGS1_Field[nItemIndex];
		IF stItem.bValidate THEN
			IF (LEN(sGS1_11) = stItem.nCodeLength OR stItem.nCodeLength = 0)  AND  ( sGS1_11 =  stGS1_AI_Definition.stAI_11.sDataField OR stGS1_AI_Definition.stAI_11.sDataField = '')  THEN
				bGS1_11_OK := TRUE;
			END_IF
		ELSE
			bGS1_11_OK := TRUE;
		END_IF
		EXIT;
	END_IF
END_FOR

(*********************** ********************************************)
(*********************** GS1_15**************************************)
bGS1_15_OK := FALSE;
sGS1_15 := F_GS1_GetItem(sFullCode, GS1_15, stCodeInfo);

FOR nItemIndex :=1 TO cMAX_VALIDATION_ITEMS DO
	IF stCodeInfo.stGS1_Field[nItemIndex].eGS1_AIType =  GS1_15 THEN
		stItem := stCodeInfo.stGS1_Field[nItemIndex];
		IF stItem.bValidate THEN
			IF( LEN(sGS1_15) = stItem.nCodeLength OR stItem.nCodeLength = 0) AND  ( sGS1_15 =  stGS1_AI_Definition.stAI_15.sDataField OR stGS1_AI_Definition.stAI_15.sDataField = '')  THEN
				bGS1_15_OK := TRUE;
			END_IF
		ELSE
			bGS1_15_OK := TRUE;
		END_IF
		EXIT;
	END_IF
END_FOR

(*********************** ********************************************)
(*********************** GS1_17**************************************)
bGS1_17_OK := FALSE;
sGS1_17 := F_GS1_GetItem(sFullCode, GS1_17, stCodeInfo);

FOR nItemIndex :=1 TO cMAX_VALIDATION_ITEMS DO
	IF stCodeInfo.stGS1_Field[nItemIndex].eGS1_AIType =  GS1_17 THEN
		stItem := stCodeInfo.stGS1_Field[nItemIndex];
		IF stItem.bValidate THEN
			IF( LEN(sGS1_17) = stItem.nCodeLength OR stItem.nCodeLength = 0) AND  ( sGS1_17 =  stGS1_AI_Definition.stAI_17.sDataField OR stGS1_AI_Definition.stAI_17.sDataField = '')  THEN
				bGS1_17_OK := TRUE;
			END_IF
		ELSE
			bGS1_17_OK := TRUE;
		END_IF
		EXIT;
	END_IF
END_FOR

(*********************** ********************************************)
(*********************** GS1_21**************************************)
bGS1_21_OK := FALSE;
sGS1_21 := F_GS1_GetItem(sFullCode, GS1_21, stCodeInfo);

FOR nItemIndex :=1 TO cMAX_VALIDATION_ITEMS DO
	IF stCodeInfo.stGS1_Field[nItemIndex].eGS1_AIType =  GS1_21 THEN
		stItem := stCodeInfo.stGS1_Field[nItemIndex];
		IF stItem.bValidate THEN
			IF( LEN(sGS1_21) = stItem.nCodeLength OR stItem.nCodeLength = 0) AND  ( sGS1_21 =  stGS1_AI_Definition.stAI_21.sDataField OR stGS1_AI_Definition.stAI_21.sDataField = '')THEN
				bGS1_21_OK := TRUE;
			END_IF
		ELSE
			bGS1_21_OK := TRUE;
		END_IF
		EXIT;
	END_IF
END_FOR

(*********************** ********************************************)
(*********************** GS1_240**************************************)
bGS1_240_OK := FALSE;
sGS1_240 := F_GS1_GetItem(sFullCode, GS1_240, stCodeInfo);

FOR nItemIndex :=1 TO cMAX_VALIDATION_ITEMS DO
	IF stCodeInfo.stGS1_Field[nItemIndex].eGS1_AIType =  GS1_240 THEN
		stItem := stCodeInfo.stGS1_Field[nItemIndex];
		IF stItem.bValidate THEN
			IF (LEN(sGS1_240) = stItem.nCodeLength OR stItem.nCodeLength = 0) AND  ( sGS1_240 =  stGS1_AI_Definition.stAI_240.sDataField OR stGS1_AI_Definition.stAI_240.sDataField = '') THEN
				bGS1_240_OK := TRUE;
			END_IF
		ELSE
			bGS1_240_OK := TRUE;
		END_IF
		EXIT;
	END_IF
END_FOR

(*********************** ********************************************)
(*********************** GS1_8005************************************)
bGS1_8005_OK := FALSE;
sGS1_8005 := F_GS1_GetItem(sFullCode, GS1_8005, stCodeInfo);

FOR nItemIndex :=1 TO cMAX_VALIDATION_ITEMS DO
	IF stCodeInfo.stGS1_Field[nItemIndex].eGS1_AIType =  GS1_8005 THEN
		stItem := stCodeInfo.stGS1_Field[nItemIndex];
		IF stItem.bValidate THEN
			IF (LEN(sGS1_8005) = stItem.nCodeLength OR stItem.nCodeLength = 0) AND  ( sGS1_8005 =  stGS1_AI_Definition.stAI_8005.sDataField OR stGS1_AI_Definition.stAI_8005.sDataField = '') THEN
				bGS1_8005_OK := TRUE;
			END_IF
		ELSE
			bGS1_8005_OK := TRUE;
		END_IF
		EXIT;
	END_IF
END_FOR

(*********************** ********************************************)
(*********************** GS1_8006************************************)
bGS1_8006_OK := FALSE;
sGS1_8006 := F_GS1_GetItem(sFullCode, GS1_8006, stCodeInfo);

FOR nItemIndex :=1 TO cMAX_VALIDATION_ITEMS DO
	IF stCodeInfo.stGS1_Field[nItemIndex].eGS1_AIType =  GS1_8006 THEN
		stItem := stCodeInfo.stGS1_Field[nItemIndex];
		IF stItem.bValidate THEN
			IF (LEN(sGS1_8006) = stItem.nCodeLength OR stItem.nCodeLength = 0) AND  ( sGS1_8006 =  stGS1_AI_Definition.stAI_8006.sDataField OR stGS1_AI_Definition.stAI_8006.sDataField = '') THEN
				bGS1_8006_OK := TRUE;
			END_IF
		ELSE
			bGS1_8006_OK := TRUE;
		END_IF
		EXIT;
	END_IF
END_FOR

(*********************** ********************************************)
(*********************** GS1_8008************************************)
bGS1_8008_OK := FALSE;
sGS1_8008 := F_GS1_GetItem(sFullCode, GS1_8008, stCodeInfo);

FOR nItemIndex :=1 TO cMAX_VALIDATION_ITEMS DO
	IF stCodeInfo.stGS1_Field[nItemIndex].eGS1_AIType =  GS1_8008 THEN
		stItem := stCodeInfo.stGS1_Field[nItemIndex];
		IF stItem.bValidate THEN
			IF (LEN(sGS1_8008) = stItem.nCodeLength OR stItem.nCodeLength = 0) AND  ( sGS1_8008 =  stGS1_AI_Definition.stAI_8008.sDataField OR stGS1_AI_Definition.stAI_8008.sDataField = '') THEN
				bGS1_8008_OK := TRUE;
			END_IF
		ELSE
			bGS1_8008_OK := TRUE;
		END_IF
		EXIT;
	END_IF
END_FOR

(*********************** ********************************************)
(*********************** GS1_91**************************************)
bGS1_91_OK := FALSE;
sGS1_91 := F_GS1_GetItem(sFullCode, GS1_91, stCodeInfo);

FOR nItemIndex :=1 TO cMAX_VALIDATION_ITEMS DO
	IF stCodeInfo.stGS1_Field[nItemIndex].eGS1_AIType =  GS1_91 THEN
		stItem := stCodeInfo.stGS1_Field[nItemIndex];
		IF stItem.bValidate THEN
			IF (LEN(sGS1_91) = stItem.nCodeLength OR stItem.nCodeLength = 0)  AND  ( sGS1_91 =  stGS1_AI_Definition.stAI_91.sDataField OR stGS1_AI_Definition.stAI_91.sDataField = '') THEN
				bGS1_91_OK := TRUE;
			END_IF
		ELSE
			bGS1_91_OK := TRUE;
		END_IF
		EXIT;
	END_IF
END_FOR

(*********************** ********************************************)
(*********************** GS1_92**************************************)
bGS1_92_OK := FALSE;
sGS1_92 := F_GS1_GetItem(sFullCode, GS1_92, stCodeInfo);

FOR nItemIndex :=1 TO cMAX_VALIDATION_ITEMS DO
	IF stCodeInfo.stGS1_Field[nItemIndex].eGS1_AIType =  GS1_92 THEN
		stItem := stCodeInfo.stGS1_Field[nItemIndex];
		IF stItem.bValidate THEN
			IF (LEN(sGS1_92) = stItem.nCodeLength OR stItem.nCodeLength = 0) AND   ( sGS1_92 =  stGS1_AI_Definition.stAI_92.sDataField OR stGS1_AI_Definition.stAI_92.sDataField = '') THEN
				bGS1_92_OK := TRUE;
			END_IF
		ELSE
			bGS1_92_OK := TRUE;
		END_IF
		EXIT;
	END_IF
END_FOR

(*********************** ********************************************)
(*********************** GS1_93**************************************)
bGS1_93_OK := FALSE;
sGS1_93 := F_GS1_GetItem(sFullCode, GS1_93, stCodeInfo);

FOR nItemIndex :=1 TO cMAX_VALIDATION_ITEMS DO
	IF stCodeInfo.stGS1_Field[nItemIndex].eGS1_AIType =  GS1_93 THEN
		stItem := stCodeInfo.stGS1_Field[nItemIndex];
		IF stItem.bValidate THEN
			IF (LEN(sGS1_93) = stItem.nCodeLength OR stItem.nCodeLength = 0)  AND  ( sGS1_93 =  stGS1_AI_Definition.stAI_93.sDataField OR stGS1_AI_Definition.stAI_93.sDataField = '') THEN
				bGS1_93_OK := TRUE;
			END_IF
		ELSE
			bGS1_93_OK := TRUE;
		END_IF
		EXIT;
	END_IF
END_FOR

(*********************** ********************************************)
(*********************** GS1_94**************************************)
bGS1_94_OK := FALSE;
sGS1_94 := F_GS1_GetItem(sFullCode, GS1_94, stCodeInfo);

FOR nItemIndex :=1 TO cMAX_VALIDATION_ITEMS DO
	IF stCodeInfo.stGS1_Field[nItemIndex].eGS1_AIType =  GS1_94 THEN
		stItem := stCodeInfo.stGS1_Field[nItemIndex];
		IF stItem.bValidate THEN
			IF (LEN(sGS1_94) = stItem.nCodeLength OR stItem.nCodeLength = 0) AND  ( sGS1_94 =  stGS1_AI_Definition.stAI_94.sDataField OR stGS1_AI_Definition.stAI_94.sDataField = '') THEN
				bGS1_94_OK := TRUE;
			END_IF
		ELSE
			bGS1_94_OK := TRUE;
		END_IF
		EXIT;
	END_IF
END_FOR

(*********************** ********************************************)

(*********************** NON_GS1_01**************************************)
bNON_GS1_01_OK := FALSE;
sNON_GS1_01 := F_GS1_GetItem(sFullCode, NON_GS1_01, stCodeInfo);

FOR nItemIndex :=1 TO cMAX_VALIDATION_ITEMS DO
	IF stCodeInfo.stGS1_Field[nItemIndex].eGS1_AIType =  NON_GS1_01 THEN
		stItem := stCodeInfo.stGS1_Field[nItemIndex];
		IF stItem.bValidate THEN
			IF (LEN(sNON_GS1_01) = stItem.nCodeLength OR stItem.nCodeLength = 0) AND  ( sNON_GS1_01 =  stGS1_AI_Definition.stNON_GS1_01.sDataField OR stGS1_AI_Definition.stNON_GS1_01.sDataField = '') THEN
				bNON_GS1_01_OK := TRUE;
			END_IF
		ELSE
			bNON_GS1_01_OK := TRUE;
		END_IF
		EXIT;
	END_IF
END_FOR

(*********************** ********************************************)
(*********************** NON_GS1_02**************************************)
bNON_GS1_02_OK := FALSE;
sNON_GS1_02 := F_GS1_GetItem(sFullCode, NON_GS1_02, stCodeInfo);

FOR nItemIndex :=1 TO cMAX_VALIDATION_ITEMS DO
	IF stCodeInfo.stGS1_Field[nItemIndex].eGS1_AIType =  NON_GS1_02 THEN
		stItem := stCodeInfo.stGS1_Field[nItemIndex];
		IF stItem.bValidate THEN
			IF (LEN(sNON_GS1_02) = stItem.nCodeLength OR stItem.nCodeLength = 0) AND  ( sNON_GS1_02 =  stGS1_AI_Definition.stNON_GS1_02.sDataField OR stGS1_AI_Definition.stNON_GS1_02.sDataField = '') THEN
				bNON_GS1_02_OK := TRUE;
			END_IF
		ELSE
			bNON_GS1_02_OK := TRUE;
		END_IF
		EXIT;
	END_IF
END_FOR

(*********************** ********************************************)
(*********************** NON_GS1_03**************************************)
bNON_GS1_03_OK := FALSE;
sNON_GS1_03 := F_GS1_GetItem(sFullCode, NON_GS1_03, stCodeInfo);

FOR nItemIndex :=1 TO cMAX_VALIDATION_ITEMS DO
	IF stCodeInfo.stGS1_Field[nItemIndex].eGS1_AIType =  NON_GS1_03 THEN
		stItem := stCodeInfo.stGS1_Field[nItemIndex];
		IF stItem.bValidate THEN
			IF (LEN(sNON_GS1_03) = stItem.nCodeLength OR stItem.nCodeLength = 0) AND  ( sNON_GS1_03 =  stGS1_AI_Definition.stNON_GS1_03.sDataField OR stGS1_AI_Definition.stNON_GS1_03.sDataField = '') THEN
				bNON_GS1_03_OK := TRUE;
			END_IF
		ELSE
			bNON_GS1_03_OK := TRUE;
		END_IF
		EXIT;
	END_IF
END_FOR

(*********************** ********************************************)
(*********************** NON_GS1_04**************************************)
bNON_GS1_04_OK := FALSE;
sNON_GS1_04 := F_GS1_GetItem(sFullCode, NON_GS1_04, stCodeInfo);

FOR nItemIndex :=1 TO cMAX_VALIDATION_ITEMS DO
	IF stCodeInfo.stGS1_Field[nItemIndex].eGS1_AIType =  NON_GS1_04 THEN
		stItem := stCodeInfo.stGS1_Field[nItemIndex];
		IF stItem.bValidate THEN
			IF (LEN(sNON_GS1_04) = stItem.nCodeLength OR stItem.nCodeLength = 0) AND  ( sNON_GS1_04 =  stGS1_AI_Definition.stNON_GS1_04.sDataField OR stGS1_AI_Definition.stNON_GS1_04.sDataField = '') THEN
				bNON_GS1_04_OK := TRUE;
			END_IF
		ELSE
			bNON_GS1_04_OK := TRUE;
		END_IF
		EXIT;
	END_IF
END_FOR

(*********************** ********************************************)
(*********************** NON_GS1_05**************************************)
bNON_GS1_05_OK := FALSE;
sNON_GS1_05 := F_GS1_GetItem(sFullCode, NON_GS1_05, stCodeInfo);

FOR nItemIndex :=1 TO cMAX_VALIDATION_ITEMS DO
	IF stCodeInfo.stGS1_Field[nItemIndex].eGS1_AIType =  NON_GS1_05 THEN
		stItem := stCodeInfo.stGS1_Field[nItemIndex];
		IF stItem.bValidate THEN
			IF (LEN(sNON_GS1_05) = stItem.nCodeLength OR stItem.nCodeLength = 0) AND  ( sNON_GS1_05 =  stGS1_AI_Definition.stNON_GS1_05.sDataField OR stGS1_AI_Definition.stNON_GS1_05.sDataField = '') THEN
				bNON_GS1_05_OK := TRUE;
			END_IF
		ELSE
			bNON_GS1_05_OK := TRUE;
		END_IF
		EXIT;
	END_IF
END_FOR

(*********************** ********************************************)
(*********************** NON_GS1_06**************************************)
bNON_GS1_06_OK := FALSE;
sNON_GS1_06 := F_GS1_GetItem(sFullCode, NON_GS1_06, stCodeInfo);

FOR nItemIndex :=1 TO cMAX_VALIDATION_ITEMS DO
	IF stCodeInfo.stGS1_Field[nItemIndex].eGS1_AIType =  NON_GS1_06 THEN
		stItem := stCodeInfo.stGS1_Field[nItemIndex];
		IF stItem.bValidate THEN
			IF (LEN(sNON_GS1_06) = stItem.nCodeLength OR stItem.nCodeLength = 0) AND  ( sNON_GS1_06 =  stGS1_AI_Definition.stNON_GS1_06.sDataField OR stGS1_AI_Definition.stNON_GS1_06.sDataField = '') THEN
				bNON_GS1_06_OK := TRUE;
			END_IF
		ELSE
			bNON_GS1_06_OK := TRUE;
		END_IF
		EXIT;
	END_IF
END_FOR

(*********************** ********************************************)
(*********************** NON_GS1_07**************************************)
bNON_GS1_07_OK := FALSE;
sNON_GS1_07 := F_GS1_GetItem(sFullCode, NON_GS1_07, stCodeInfo);

FOR nItemIndex :=1 TO cMAX_VALIDATION_ITEMS DO
	IF stCodeInfo.stGS1_Field[nItemIndex].eGS1_AIType =  NON_GS1_07 THEN
		stItem := stCodeInfo.stGS1_Field[nItemIndex];
		IF stItem.bValidate THEN
			IF (LEN(sNON_GS1_07) = stItem.nCodeLength OR stItem.nCodeLength = 0) AND  ( sNON_GS1_07 =  stGS1_AI_Definition.stNON_GS1_07.sDataField OR stGS1_AI_Definition.stNON_GS1_07.sDataField = '') THEN
				bNON_GS1_07_OK := TRUE;
			END_IF
		ELSE
			bNON_GS1_07_OK := TRUE;
		END_IF
		EXIT;
	END_IF
END_FOR

(*********************** ********************************************)
(*********************** NON_GS1_08**************************************)
bNON_GS1_08_OK := FALSE;
sNON_GS1_08 := F_GS1_GetItem(sFullCode, NON_GS1_08, stCodeInfo);

FOR nItemIndex :=1 TO cMAX_VALIDATION_ITEMS DO
	IF stCodeInfo.stGS1_Field[nItemIndex].eGS1_AIType =  NON_GS1_08 THEN
		stItem := stCodeInfo.stGS1_Field[nItemIndex];
		IF stItem.bValidate THEN
			IF (LEN(sNON_GS1_08) = stItem.nCodeLength OR stItem.nCodeLength = 0) AND  ( sNON_GS1_08 =  stGS1_AI_Definition.stNON_GS1_08.sDataField OR stGS1_AI_Definition.stNON_GS1_08.sDataField = '') THEN
				bNON_GS1_08_OK := TRUE;
			END_IF
		ELSE
			bNON_GS1_08_OK := TRUE;
		END_IF
		EXIT;
	END_IF
END_FOR

(*********************** ********************************************)
(*********************** NON_GS1_09**************************************)
bNON_GS1_09_OK := FALSE;
sNON_GS1_09 := F_GS1_GetItem(sFullCode, NON_GS1_09, stCodeInfo);

FOR nItemIndex :=1 TO cMAX_VALIDATION_ITEMS DO
	IF stCodeInfo.stGS1_Field[nItemIndex].eGS1_AIType =  NON_GS1_09 THEN
		stItem := stCodeInfo.stGS1_Field[nItemIndex];
		IF stItem.bValidate THEN
			IF (LEN(sNON_GS1_09) = stItem.nCodeLength OR stItem.nCodeLength = 0) AND  ( sNON_GS1_09 =  stGS1_AI_Definition.stNON_GS1_09.sDataField OR stGS1_AI_Definition.stNON_GS1_09.sDataField = '') THEN
				bNON_GS1_09_OK := TRUE;
			END_IF
		ELSE
			bNON_GS1_09_OK := TRUE;
		END_IF
		EXIT;
	END_IF
END_FOR

(*********************** ********************************************)
(*********************** NON_GS1_10**************************************)
bNON_GS1_10_OK := FALSE;
sNON_GS1_10 := F_GS1_GetItem(sFullCode, NON_GS1_10, stCodeInfo);

FOR nItemIndex :=1 TO cMAX_VALIDATION_ITEMS DO
	IF stCodeInfo.stGS1_Field[nItemIndex].eGS1_AIType =  NON_GS1_10 THEN
		stItem := stCodeInfo.stGS1_Field[nItemIndex];
		IF stItem.bValidate THEN
			IF (LEN(sNON_GS1_10) = stItem.nCodeLength OR stItem.nCodeLength = 0) AND  ( sNON_GS1_10 =  stGS1_AI_Definition.stNON_GS1_10.sDataField OR stGS1_AI_Definition.stNON_GS1_10.sDataField = '') THEN
				bNON_GS1_10_OK := TRUE;
			END_IF
		ELSE
			bNON_GS1_10_OK := TRUE;
		END_IF
		EXIT;
	END_IF
END_FOR

(*********************** ********************************************)


bValidationOK	:= bEntireCodeLengthOK;

FOR nItemIndex :=1 TO cMAX_VALIDATION_ITEMS DO
	CASE stCodeInfo.stGS1_Field[nItemIndex].eGS1_AIType OF
	GS1_01:
		bValidationOK := bValidationOK AND bGS1_01_OK;
	GS1_10:
		bValidationOK := bValidationOK AND bGS1_10_OK;
	GS1_11:
		bValidationOK := bValidationOK AND bGS1_11_OK;
	GS1_15:
		bValidationOK := bValidationOK AND bGS1_15_OK;
	GS1_17:
		bValidationOK := bValidationOK AND bGS1_17_OK;
	GS1_21:
		bValidationOK := bValidationOK AND bGS1_21_OK;
	GS1_240:
		bValidationOK := bValidationOK AND bGS1_240_OK;
	GS1_8005:
		bValidationOK := bValidationOK AND bGS1_8005_OK;
	GS1_8006:
		bValidationOK := bValidationOK AND bGS1_8006_OK;
	GS1_8008:
		bValidationOK := bValidationOK AND bGS1_8008_OK;
	GS1_91:
		bValidationOK := bValidationOK AND bGS1_91_OK;
	GS1_92:
		bValidationOK := bValidationOK AND bGS1_92_OK;
	GS1_93:
		bValidationOK := bValidationOK AND bGS1_93_OK;
	GS1_94:
		bValidationOK := bValidationOK AND bGS1_94_OK;
	NON_GS1_01:
		bValidationOK := bValidationOK AND bNON_GS1_01_OK;
	NON_GS1_02:
		bValidationOK := bValidationOK AND bNON_GS1_02_OK;
	NON_GS1_03:
		bValidationOK := bValidationOK AND bNON_GS1_03_OK;
	NON_GS1_04:
		bValidationOK := bValidationOK AND bNON_GS1_04_OK;
	NON_GS1_05:
		bValidationOK := bValidationOK AND bNON_GS1_05_OK;
	NON_GS1_06:
		bValidationOK := bValidationOK AND bNON_GS1_06_OK;
	NON_GS1_07:
		bValidationOK := bValidationOK AND bNON_GS1_07_OK;
	NON_GS1_08:
		bValidationOK := bValidationOK AND bNON_GS1_08_OK;
	NON_GS1_09:
		bValidationOK := bValidationOK AND bNON_GS1_09_OK;
	NON_GS1_10:
		bValidationOK := bValidationOK AND bNON_GS1_10_OK;
	END_CASE
END_FOR

END_FUNCTION_BLOCK

// ---- POUs/_Utilites/METS/Common LIB/08_SOFTWARE LIB/AI GS1 Codes And Validation FBs/F_GS1_GetItem.TcPOU
FUNCTION F_GS1_GetItem : T_MaxString
VAR_INPUT
	sFullCode			: T_MaxString;
	eCodeAIType		: E_GS1_CodeAIType;
	stCodeInfo		: ST_GS1_CodeInfo;
END_VAR
VAR
	stItem			: ST_GS1_CodeValidation;
	nItemIndex		: INT;
	(*eCodeAIPattern	: E_CodeAIType;*)
	sItem			: T_MaxString;
	nStart			: INT;
	nEnd				: INT;
	sTemp			: T_MaxString;
END_VAR

IF stCodeInfo.nEntireLength > 0 THEN

	FOR nItemIndex :=1 TO cMAX_VALIDATION_ITEMS DO
		IF eCodeAIType = stCodeInfo.stGS1_Field[nItemIndex].eGS1_AIType THEN
			stItem := stCodeInfo.stGS1_Field[nItemIndex];
			EXIT;
		ELSE
			F_GS1_GetItem := 'Validation Item Not Found';
		END_IF
	END_FOR


	IF stItem.sStartAI <> '' AND stItem.sEndAI <> '' THEN
		nStart := FIND(sFullCode, stItem.sStartAI) + LEN(stItem.sStartAI);
		IF nStart > 0 THEN
			sTemp := RIGHT(sFullCode, LEN(sFullCode) - (nStart - 1));
		ELSE
			sTemp := sFullCode;
		END_IF
		nEnd := FIND(sTemp, stItem.sEndAI);
		IF nEnd = 0 THEN
			nEnd := LEN(sFullCode)+1;
		ELSE
			nEnd := nEnd +(nStart - 1);
		END_IF
	ELSIF stItem.sStartAI <> '' AND stItem.nCodeLength > 0 THEN
		nStart := FIND(sFullCode, stItem.sStartAI) + LEN(stItem.sStartAI);
		nEnd := nStart + stItem.nCodeLength;
	ELSIF stItem.nCodeStartPos > 0 AND stItem.sEndAI <> '' THEN
		nStart := stItem.nCodeStartPos;
		sTemp := RIGHT(sFullCode, LEN(sFullCode) - (nStart - 1));
		nEnd := FIND(sTemp, stItem.sEndAI);
		IF nEnd = 0 THEN
			nEnd := LEN(sFullCode)+1;
		ELSE
			nEnd := nEnd +(nStart - 1);
		END_IF
	ELSIF stItem.nCodeStartPos >= 0 AND stItem.nCodeLength > 0 THEN
		nStart := stItem.nCodeStartPos;
		nEnd := nStart + stItem.nCodeLength;
	ELSE
		nStart := 0;
		nEnd := 0;
	END_IF
	IF nStart > 0 AND nEnd > 0 THEN
		sItem := MID(sFullCode, nEnd - nStart, nStart);
	ELSE
		sItem := '';
	END_IF
ELSE
	sItem := '';
END_IF

F_GS1_GetItem := sItem;

END_FUNCTION

// ---- POUs/_Utilites/METS/Concat Function/F_CONCAT7.TcPOU
(* concatenate 7 strings *)
FUNCTION F_CONCAT7 : T_MaxString
VAR_INPUT
	strString1		: T_MaxString;
	strString2		: T_MaxString;
	strString3		: T_MaxString;
	strString4		: T_MaxString;
	strString5		: T_MaxString;
	strString6		: T_MaxString;
	strString7		: T_MaxString;
END_VAR
VAR
END_VAR
(*
-------------------------------------------------------------------------------------------------
Date		Version	Author	Comments
-------------------------------------------------------------------------------------------------
30/01/2015	3.00.00	PB		No change

-------------------------------------------------------------------------------------------------
05/02/2010	1.00.00	PB		Initial release

-------------------------------------------------------------------------------------------------
*)

F_CONCAT7 := CONCAT(strString1, strString2);
F_CONCAT7 := CONCAT(F_CONCAT7, strString3);
F_CONCAT7 := CONCAT(F_CONCAT7, strString4);
F_CONCAT7 := CONCAT(F_CONCAT7, strString5);
F_CONCAT7 := CONCAT(F_CONCAT7, strString6);
F_CONCAT7 := CONCAT(F_CONCAT7, strString7);

END_FUNCTION

// ---- POUs/_Utilites/METS/Concat Function/F_CONCAT8.TcPOU
(* concatenate 8 strings *)
FUNCTION F_CONCAT8 : T_MaxString
VAR_INPUT
	strString1		: T_MaxString;
	strString2		: T_MaxString;
	strString3		: T_MaxString;
	strString4		: T_MaxString;
	strString5		: T_MaxString;
	strString6		: T_MaxString;
	strString7		: T_MaxString;
	strString8		: T_MaxString;
END_VAR
VAR
END_VAR
(*
-------------------------------------------------------------------------------------------------
Date		Version	Author	Comments
-------------------------------------------------------------------------------------------------
30/01/2015	3.00.00	PB		No change

-------------------------------------------------------------------------------------------------
05/02/2010	1.00.00	PB		Initial release

-------------------------------------------------------------------------------------------------
*)

F_CONCAT8 := CONCAT(strString1, strString2);
F_CONCAT8 := CONCAT(F_CONCAT8, strString3);
F_CONCAT8 := CONCAT(F_CONCAT8, strString4);
F_CONCAT8 := CONCAT(F_CONCAT8, strString5);
F_CONCAT8 := CONCAT(F_CONCAT8, strString6);
F_CONCAT8 := CONCAT(F_CONCAT8, strString7);
F_CONCAT8 := CONCAT(F_CONCAT8, strString8);

END_FUNCTION

// ---- POUs/_Utilites/METS/Concat Function/F_CONCAT9.TcPOU
(* concatenate 9 strings *)
FUNCTION F_CONCAT9 : T_MaxString
VAR_INPUT
	strString1		: T_MaxString;
	strString2		: T_MaxString;
	strString3		: T_MaxString;
	strString4		: T_MaxString;
	strString5		: T_MaxString;
	strString6		: T_MaxString;
	strString7		: T_MaxString;
	strString8		: T_MaxString;
	strString9		: T_MaxString;
END_VAR
VAR
END_VAR
(*
-------------------------------------------------------------------------------------------------
Date		Version	Author	Comments
-------------------------------------------------------------------------------------------------
30/01/2015	3.00.00	PB		No change

-------------------------------------------------------------------------------------------------
05/02/2010	1.00.00	PB		Initial release

-------------------------------------------------------------------------------------------------
*)

F_CONCAT9 := CONCAT(strString1, strString2);
F_CONCAT9 := CONCAT(F_CONCAT9, strString3);
F_CONCAT9 := CONCAT(F_CONCAT9, strString4);
F_CONCAT9 := CONCAT(F_CONCAT9, strString5);
F_CONCAT9 := CONCAT(F_CONCAT9, strString6);
F_CONCAT9 := CONCAT(F_CONCAT9, strString7);
F_CONCAT9 := CONCAT(F_CONCAT9, strString8);
F_CONCAT9 := CONCAT(F_CONCAT9, strString9);

END_FUNCTION

// ---- POUs/_Utilites/METS/F_CASE_GetSKUFromHex.TcPOU
FUNCTION F_CASE_GetSKUFromHex : STRING(8)
VAR_INPUT
	sSKU_FromCase	: STRING(7);
END_VAR
VAR

	nSKULen			: INT;
	nCharIndex		: INT;
	strChar				: STRING(1);
	nCharInDec		: REAL;
	nData				: lREAL;
	sSKU_Number		: STRING;

END_VAR

(* reset output *)
F_CASE_GetSKUFromHex := '';


(* length of strPackCode *)
nSKULen := LEN(sSKU_FromCase);
nData:=0;
(* strPackCode contains data *)
IF nSKULen > 0 THEN

	(* check each char in the code *)
	FOR nCharIndex := 1 TO nSKULen DO
		(* get char from string *)
		strChar := MID(sSKU_FromCase, 1, nCharIndex);
		nCharInDec := BYTE_TO_INT(HEXCHRNIBBLE_TO_BYTE(strChar));
		nData:= nCharInDec*EXPT(16,nSKULen-nCharIndex) + nData;
	END_FOR
END_IF

F_CASE_GetSKUFromHex := LEFT(lREAL_TO_STRING(nData),8);

END_FUNCTION

// ---- POUs/_Utilites/METS/F_SafeDIV.TcPOU
(* F_SafeDiv prevents PLC crash with DIV0 error by pre-checking that the denominator <> 0 *)
(* Value of 0 is returned if denominator = 0 *)
FUNCTION F_SafeDIV : LREAL
VAR_INPUT
	fNumerator		: LREAL;
	fDenominator	: LREAL;
END_VAR
(*
-------------------------------------------------------------------------------------------------
Date		Version	Author	Comments
-------------------------------------------------------------------------------------------------
30/01/2015	3.00.00	PB		LREAL now used in place of REAL

-------------------------------------------------------------------------------------------------
05/02/10	1.00.00	PB		Initial release

-------------------------------------------------------------------------------------------------
*)

(* do not perform DIV if Denominator = 0 *)
IF fDenominator = 0 THEN

	F_SafeDIV := 0;

(* safe to perform DIV *)
ELSE

	F_SafeDIV := fNumerator / fDenominator;
END_IF

END_FUNCTION

// ---- POUs/_Utilites/METS/F_ZeroPadString.TcPOU
(* append leading zeroes to a string to make up to specified length, max 19 chars *)
FUNCTION F_ZeroPadString : STRING(19)
VAR_INPUT
	strString		: STRING(19);	(* initial string *)
	nPadLength 		: BYTE;		(* string length required *)
END_VAR
VAR
	nMaxLength		: BYTE;
END_VAR
(*
-------------------------------------------------------------------------------------------------
Date		Version	Author	Comments
-------------------------------------------------------------------------------------------------
03/08/2012	1.39.00	PB		String lengths reduced to 19 characters.
							Trap added to prevent PLC from crashing if nPadLength > 19.
12/11/2010	1.07.00	PB		Initial release

-------------------------------------------------------------------------------------------------
*)

(* max string length *)
nMaxLength := SIZEOF(F_ZeroPadString) - 1;

(* initial string *)
F_ZeroPadString := strString;

(* string length is shorter than required/max length *)
WHILE LEN(F_ZeroPadString) < MIN(nPadLength, nMaxLength) DO

	(* append leading '0' char to string *)
	F_ZeroPadString := CONCAT('0', F_ZeroPadString);
END_WHILE

END_FUNCTION

// ---- POUs/_Utilites/Tests/FB_FIND_OuterDuplicates.TcPOU
FUNCTION_BLOCK FB_FIND_OuterDuplicates
VAR_INPUT
END_VAR
VAR_OUTPUT
	bHasDuplicates		: BOOL;
	nDuplicateCount		: UINT;
	nIterationCount		: UINT;
END_VAR
VAR
	nOuterIndex			: UINT;
	nInnerOuterIndex	: UINT;
	nInnerPackIndex		: UINT;
	nPackIndex			: UINT;
	sCurrentOuterCode	: T_MaxString;
	sCurrentPackCode	: T_MaxString;	
	bIsDuplicate 		: BOOL;
	bISOuterDuplicate	: BOOL;
END_VAR
VAR_IN_OUT	
	stCase				: ST_LAB_CaseData;
END_VAR


bHasDuplicates := FALSE;
nDuplicateCount := 0;
	
	(* Loop throught all packs in one case 'stCase' *)
	FOR nOuterIndex := 1 TO GVL_test.nMax_Outers DO
		sCurrentOuterCode := stCase.aOuters[nOuterIndex].sOuterCode;
		FOR nPackIndex := 1 TO GVL_test.nMax_Packs DO
			sCurrentPackCode := stCase.aOuters[nOuterIndex].aPacks[nPackIndex].sPackCode;
			bIsDuplicate := FALSE;			
			(* Looking for same pack codes in all outers *)
			FOR nInnerOuterIndex := nOuterIndex TO GVL_test.nMax_Outers DO
				IF nInnerOuterIndex < 50 THEN					
					IF (sCurrentOuterCode = stCase.aOuters[nInnerOuterIndex + 1].sOuterCode) THEN
						bIsOuterDuplicate									:= TRUE;													
						stCase.aOuters[nOuterIndex].nOuterRejectID			:= 200;					
						stCase.aOuters[nInnerOuterIndex + 1].nOuterRejectID	:= 200;
					END_IF	
				END_IF
				FOR nInnerPackIndex := 1 TO GVL_test.nMax_Packs DO
					nIterationCount	:= nIterationCount + 1;					
					(* Exclude comparing same pack with itself *)
					IF NOT ((nInnerOuterIndex = nOuterIndex) AND (nInnerPackIndex = nPackIndex)) THEN
						IF sCurrentPackCode = stCase.aOuters[nInnerOuterIndex].aPacks[nInnerPackIndex].sPackCode THEN
							bIsDuplicate := TRUE;
							nDuplicateCount := nDuplicateCount + 1;
							
							stCase.aOuters[nInnerOuterIndex].aPacks[nInnerPackIndex].nPackRejectID	:= 200;
							stCase.aOuters[nInnerOuterIndex].nOuterRejectID							:= 200;
							
							stCase.aOuters[nOuterIndex].aPacks[nPackIndex].nPackRejectID			:= 200;
							stCase.aOuters[nOuterIndex].nOuterRejectID								:= 200;
						END_IF
					END_IF
				END_FOR
			END_FOR			
			IF bIsDuplicate THEN
				bHasDuplicates 	:= TRUE;
			END_IF
		END_FOR
	END_FOR
	
	
	(* nDuplicateCount includes all elements with same pack codes *)
	(* the number of duplicated codes is nDuplicateCount/2 *)

END_FUNCTION_BLOCK

// ---- POUs/_Utilites/Tests/FB_FIND_OuterDuplicatesPiotr.TcPOU
FUNCTION_BLOCK FB_FIND_OuterDuplicatesPiotr
VAR_INPUT
	bExecute	: BOOL;
END_VAR
VAR_IN_OUT

	//stProductInstruction				: ST_PCM_Status;
	
	//stPackCodesDuplicated			: ST_RejectItems;
	//stOuterBarcodeDuplicate			: ST_RejectItems;
	//stOuterDuplicatedPackCodesFound	: ST_RejectItems;
	//stCaseRejectReasons			: ST_RejectReasonsForCase;
	
	//stCACData 						: ST_CAC_Data;
	
	(* for AI mode*)	
	stCase				: ST_LAB_CaseData;
	
END_VAR
VAR_OUTPUT
	//bDone 					: BOOL;
	//bBusy					: BOOL;

	//bCACValid				: BOOL;
	//sRejectCode				: T_MaxString;
	//bIsDuplicateOuters		: BOOL;
	//bIsDuplicatePacks		: BOOL;
END_VAR
VAR

	rtExecute	: R_TRIG;
	
	nOuterIndex			: UINT;
	nPackIndex			: UINT;
	//nOuterCheckIndex	: INT;
	nInnerOuterIndex	: UINT;
	//nPackCheckIndex		: INT;
	nInnerPackIndex		: UINT;
	
	nDuplicateOuter1_Position	: UINT;
	nDuplicateOuter2_Position	: UINT;
	nDuplicatePack1_Position	: UINT;
	nDuplicatePack2_Position	: UINT;
	
	aStatusErrorVal					: ARRAY[0..10] OF STRING(10);
	aRejectCodePointer     		   	: ARRAY[0..10] OF STRING(10);
	
	nIteration				: UDINT;
	nIterationAI			: UDINT;
	
	bIsDuplicateOuters		: BOOL;
	bIsDuplicatePacks		: BOOL;
END_VAR

rtExecute(CLK:=bExecute);

IF rtExecute.Q THEN
	
	(* update outputs *)
	//bDone := TRUE;
	//bBusy := TRUE;

	bIsDuplicateOuters:= FALSE;
	bIsDuplicatePacks:= FALSE;
	
	MEMSET(ADR(aStatusErrorVal), 16#00, SIZEOF(aStatusErrorVal));
	MEMSET(ADR(aRejectCodePointer), 16#00, SIZEOF(aRejectCodePointer));

	nDuplicateOuter1_Position :=0;
	nDuplicateOuter2_Position:=0;
	nDuplicatePack1_Position:=0;
	nDuplicatePack2_Position:=0;

	(* clear outputs *)
	//bCACValid := FALSE;
	//sRejectCode := '';
	
	nIteration		:= 0;
	nIterationAI	:= 0;
	
	
//////////////////////	
	FOR nOuterIndex := 1 TO GVL_test.nMax_Outers BY 1 DO
	//////////////////////		
		FOR nInnerOuterIndex := nOuterIndex + 1 TO GVL_test.nMax_Outers BY 1 DO
			
			IF stCase.aOuters[nOuterIndex].sOuterCode = stCase.aOuters[nInnerOuterIndex].sOuterCode AND 
				stCase.aOuters[nOuterIndex].sOuterCode <> ''	THEN
				 
			 	IF NOT bIsDuplicateOuters THEN
					nDuplicateOuter1_Position := nOuterIndex;
					nDuplicateOuter2_Position := nInnerOuterIndex;
				END_IF
					
				bIsDuplicateOuters := TRUE; 
				
				stCase.aOuters[nOuterIndex].nOuterRejectID			:=	200;
				stCase.aOuters[nInnerOuterIndex].nOuterRejectID		:=	200;
			 END_IF
			 nIteration := nIteration + 1;
		END_FOR
		///////////////////////////
		FOR  nPackIndex :=1 TO GVL_test.nMax_Packs BY 1 DO
			FOR nInnerPackIndex := nPackIndex + 1  TO GVL_test.nMax_Packs BY 1 DO
				
				IF stCase.aOuters[nOuterIndex].aPacks[nPackIndex].sPackCode = stCase.aOuters[nOuterIndex].aPacks[nInnerPackIndex].sPackCode AND 
					stCase.aOuters[nOuterIndex].aPacks[nPackIndex].sPackCode  <> ''										AND 
					stCase.aOuters[nOuterIndex].aPacks[nInnerPackIndex].nPackStatus <> 200 	THEN
					
					IF NOT bIsDuplicatePacks AND NOT bIsDuplicateOuters THEN
						nDuplicateOuter1_Position := nOuterIndex;
						nDuplicateOuter2_Position :=  nOuterIndex;
						nDuplicatePack1_Position := nPackIndex;
						nDuplicatePack2_Position := nInnerPackIndex;
					END_IF
						
					bIsDuplicatePacks := TRUE;
					stCase.aOuters[nOuterIndex].nOuterRejectID		:= 200;					
					stCase.aOuters[nOuterIndex].aPacks[nPackIndex].nPackRejectID		:= 200;
					stCase.aOuters[nOuterIndex].aPacks[nInnerPackIndex].nPackRejectID	:= 200;
				END_IF
				nIteration := nIteration + 1;
			END_FOR
			/////////////////////////////////
			FOR nInnerOuterIndex := nOuterIndex + 1 TO GVL_test.nMax_Outers BY 1 DO
				FOR nInnerPackIndex := 1  TO GVL_test.nMax_Packs BY 1 DO

					IF stCase.aOuters[nOuterIndex].aPacks[nPackIndex].sPackCode = stCase.aOuters[nInnerOuterIndex].aPacks[nInnerPackIndex].sPackCode AND 
						stCase.aOuters[nOuterIndex].aPacks[nPackIndex].sPackCode  <> ''									AND 
						stCase.aOuters[nInnerOuterIndex].aPacks[nInnerPackIndex].nPackRejectID <> 200 	THEN
						
						IF NOT bIsDuplicatePacks AND NOT bIsDuplicateOuters THEN
							nDuplicateOuter1_Position := nOuterIndex;
							nDuplicateOuter2_Position :=  nInnerOuterIndex;
							nDuplicatePack1_Position := nPackIndex;
							nDuplicatePack2_Position := nInnerPackIndex;
						END_IF
							
						bIsDuplicatePacks := TRUE;
						stCase.aOuters[nOuterIndex].nOuterRejectID			:= 200;						
						stCase.aOuters[nInnerOuterIndex].nOuterRejectID		:= 200;
						
						stCase.aOuters[nOuterIndex].aPacks[nPackIndex].nPackRejectID			:= 200;
						stCase.aOuters[nInnerOuterIndex].aPacks[nInnerPackIndex].nPackRejectID	:= 200;
					END_IF
					nIteration := nIteration + 1;
				END_FOR
			END_FOR
		/////////////////////////////////		
		END_FOR
	//////////////////////	
	END_FOR
//////////////////////	


	
ELSIF bExecute = FALSE THEN
	
	(* clear outputs *)
	//bDone := FALSE;
	//bBusy := FALSE;
	;

END_IF

END_FUNCTION_BLOCK

// ---- POUs/_Utilites/Tests/FB_FIND_OuterDuplicatesPiotrAI.TcPOU
FUNCTION_BLOCK FB_FIND_OuterDuplicatesPiotrAI
VAR_INPUT
END_VAR
VAR_OUTPUT
END_VAR
VAR
	nOuterIndex			: UINT;
	nInnerOuterIndex	: UINT;
	nInnerPackIndex		: UINT;
	nPackIndex			: UINT;
	sCurrentOuterCode	: T_MaxString;
	sCurrentPackCode	: T_MaxString;	
	bIsDuplicate 		: BOOL;
	bISOuterDuplicate	: BOOL;
	bIsDuplicateOuters	: BOOL;
	nIterationAI		: UINT;
	bIsDuplicatePacks	: BOOL;
END_VAR

VAR_IN_OUT	
	stCase				: ST_LAB_CaseData;
END_VAR

(* Loop throught all packs in one case 'stCase' *)
	FOR nOuterIndex := 1 TO GVL_test.nMax_Outers BY 1 DO
		FOR nPackIndex := 1 TO GVL_test.nMax_Packs BY 1 DO			
			(* Looking for same pack codes in all outers *)
			FOR nInnerOuterIndex := nOuterIndex TO GVL_test.nMax_Outers BY 1 DO
				
				IF stCase.aOuters[nOuterIndex].sOuterCode = stCase.aOuters[nInnerOuterIndex].sOuterCode AND 
					stCase.aOuters[nOuterIndex].sOuterCode <> ''										AND 
					NOT (nInnerOuterIndex = nOuterIndex) 											THEN
				 
						
					bIsDuplicateOuters := TRUE; 
					
					stCase.aOuters[nOuterIndex].nOuterRejectID			:=	200;		
					stCase.aOuters[nInnerOuterIndex].nOuterRejectID		:=	200;
				END_IF
				
				FOR nInnerPackIndex := 1 TO GVL_test.nMax_Packs BY 1 DO
					nIterationAI := nIterationAI + 1;					
					(* Exclude comparing same pack with itself *)
					IF stCase.aOuters[nOuterIndex].aPacks[nPackIndex].sPackCode = stCase.aOuters[nInnerOuterIndex].aPacks[nInnerPackIndex].sPackCode 	AND 
						stCase.aOuters[nOuterIndex].aPacks[nPackIndex].sPackCode  <> ''														AND 
						stCase.aOuters[nInnerOuterIndex].aPacks[nInnerPackIndex].nPackRejectID <> 200 				AND 
						NOT ((nInnerOuterIndex = nOuterIndex) AND (nInnerPackIndex = nPackIndex)) 										THEN
							
						bIsDuplicatePacks := TRUE;
						stCase.aOuters[nOuterIndex].nOuterRejectID		:= 200;						
						stCase.aOuters[nInnerOuterIndex].nOuterRejectID	:= 200;
						
						stCase.aOuters[nOuterIndex].aPacks[nPackIndex].nPackRejectID			:= 200;
						stCase.aOuters[nInnerOuterIndex].aPacks[nInnerPackIndex].nPackRejectID	:= 200;
					END_IF
				END_FOR
			END_FOR			
		END_FOR
	END_FOR

END_FUNCTION_BLOCK

// ---- POUs/_Utilites/Tests/IO_logic.TcPOU
PROGRAM IO_logic
VAR
	rtrigCameraTrigger			: R_TRIG;
	tTimerCameraTrigger			: TOF;
	tTrigerTime					: time := T#5ms;
END_VAR


rtrigCameraTrigger(CLK := gvl.bTriggerButton);

tTimerCameraTrigger(IN:= rtrigCameraTrigger.Q, PT:= tTrigerTime);
GVL.bTriggerOutput := tTimerCameraTrigger.Q;

END_PROGRAM

// ---- POUs/_Utilites/Tests/Outer_IN_Case_Duplicat.TcPOU
PROGRAM Outer_IN_Case_Duplicat
VAR
		
	fbFIND_OuterDuplicates			: FB_FIND_OuterDuplicates;
	fbFIND_OuterDuplicatesPiotr		: FB_FIND_OuterDuplicatesPiotr;	
	fbFIND_OuterDuplicatesPiotrAI	: FB_FIND_OuterDuplicatesPiotrAI;
	
	bHasDuplicates				: BOOL;
	nDuplicateCount				: UINT;
	
	rTrigAI						: R_TRIG;
	rTrigPiotr					: R_TRIG;
	rTrigPiotrAI					: R_TRIG;
	bExecuteAI					: BOOL;
	bExecutePiotr				: BOOL;
	
	bExecutePiotrAI				: BOOL;
	
	
	// dla petli for dla stworzenia outerow 
	rTrigDataFill	: R_TRIG;
	bDataFill		: BOOL;
	
	iOuter		: UINT;
	iPack		: UINT;
	
	sPackNum	: STRING;
	sOuterNum	: STRING;
	sPackCode	: STRING;
	
END_VAR


//CaseDataAdd();
//Case50outersADD();

FullFilOuter();

rTrigAI(CLK := bExecuteAI);

IF rTrigAI.Q THEN	
	fbFIND_OuterDuplicates(
		stCase 			:= GVL_test.stCaseFull, 
		bHasDuplicates 	=> bHasDuplicates, 
		nDuplicateCount => nDuplicateCount
	);	
	
END_IF

	
	fbFIND_OuterDuplicatesPiotr(
		bExecute := bExecutePiotr,
		stCase := GVL_test.stCaseFull		
	);

rTrigPiotrAI(CLK := bExecutePiotrAI);

IF rTrigPiotrAI.Q THEN	
	fbFIND_OuterDuplicatesPiotrAI(
		stCase := GVL_test.stCaseFull
	);	
	
END_IF

ACTION Case50outersADD:
(* ===== OUTER 1 ===== *)
GVL_test.stCase.aOuters[1].sOuterCode    := 'OUTER1';
GVL_test.stCase.aOuters[1].nOutersStatus := 5;
// packs 1..10
GVL_test.stCase.aOuters[1].aPacks[1].sPackCode   := 'PACK01OUTER1';
GVL_test.stCase.aOuters[1].aPacks[1].nPackStatus := 5;
GVL_test.stCase.aOuters[1].aPacks[2].sPackCode   := 'PACK02OUTER1';
GVL_test.stCase.aOuters[1].aPacks[2].nPackStatus := 5;
GVL_test.stCase.aOuters[1].aPacks[3].sPackCode   := 'PACK03OUTER1';
GVL_test.stCase.aOuters[1].aPacks[3].nPackStatus := 5;
GVL_test.stCase.aOuters[1].aPacks[4].sPackCode   := 'PACK04OUTER1';
GVL_test.stCase.aOuters[1].aPacks[4].nPackStatus := 5;
GVL_test.stCase.aOuters[1].aPacks[5].sPackCode   := 'PACK05OUTER1';
GVL_test.stCase.aOuters[1].aPacks[5].nPackStatus := 5;
GVL_test.stCase.aOuters[1].aPacks[6].sPackCode   := 'PACK06OUTER1';
GVL_test.stCase.aOuters[1].aPacks[6].nPackStatus := 5;
GVL_test.stCase.aOuters[1].aPacks[7].sPackCode   := 'PACK07OUTER1';
GVL_test.stCase.aOuters[1].aPacks[7].nPackStatus := 5;
GVL_test.stCase.aOuters[1].aPacks[8].sPackCode   := 'PACK08OUTER1';
GVL_test.stCase.aOuters[1].aPacks[8].nPackStatus := 5;
GVL_test.stCase.aOuters[1].aPacks[9].sPackCode   := 'PACK09OUTER1';
GVL_test.stCase.aOuters[1].aPacks[9].nPackStatus := 5;
GVL_test.stCase.aOuters[1].aPacks[10].sPackCode  := 'PACK10OUTER1';
GVL_test.stCase.aOuters[1].aPacks[10].nPackStatus := 5;

(* ===== OUTER 2 ===== *)
GVL_test.stCase.aOuters[2].sOuterCode    := 'OUTER2';
GVL_test.stCase.aOuters[2].nOutersStatus := 5;
// packs 1..10
GVL_test.stCase.aOuters[2].aPacks[1].sPackCode   := 'PACK01OUTER2';
GVL_test.stCase.aOuters[2].aPacks[1].nPackStatus := 5;
GVL_test.stCase.aOuters[2].aPacks[2].sPackCode   := 'PACK02OUTER2';
GVL_test.stCase.aOuters[2].aPacks[2].nPackStatus := 5;
GVL_test.stCase.aOuters[2].aPacks[3].sPackCode   := 'PACK03OUTER2';
GVL_test.stCase.aOuters[2].aPacks[3].nPackStatus := 5;
GVL_test.stCase.aOuters[2].aPacks[4].sPackCode   := 'PACK04OUTER2';
GVL_test.stCase.aOuters[2].aPacks[4].nPackStatus := 5;
GVL_test.stCase.aOuters[2].aPacks[5].sPackCode   := 'PACK05OUTER2';
GVL_test.stCase.aOuters[2].aPacks[5].nPackStatus := 5;
GVL_test.stCase.aOuters[2].aPacks[6].sPackCode   := 'PACK06OUTER2';
GVL_test.stCase.aOuters[2].aPacks[6].nPackStatus := 5;
GVL_test.stCase.aOuters[2].aPacks[7].sPackCode   := 'PACK07OUTER2';
GVL_test.stCase.aOuters[2].aPacks[7].nPackStatus := 5;
GVL_test.stCase.aOuters[2].aPacks[8].sPackCode   := 'PACK08OUTER2';
GVL_test.stCase.aOuters[2].aPacks[8].nPackStatus := 5;
GVL_test.stCase.aOuters[2].aPacks[9].sPackCode   := 'PACK09OUTER2';
GVL_test.stCase.aOuters[2].aPacks[9].nPackStatus := 5;
GVL_test.stCase.aOuters[2].aPacks[10].sPackCode  := 'PACK10OUTER2';
GVL_test.stCase.aOuters[2].aPacks[10].nPackStatus := 5;

(* ===== OUTER 3 ===== *)
GVL_test.stCase.aOuters[3].sOuterCode    := 'OUTER3';
GVL_test.stCase.aOuters[3].nOutersStatus := 5;
// packs 1..10
GVL_test.stCase.aOuters[3].aPacks[1].sPackCode   := 'PACK01OUTER3';
GVL_test.stCase.aOuters[3].aPacks[1].nPackStatus := 5;
GVL_test.stCase.aOuters[3].aPacks[2].sPackCode   := 'PACK02OUTER3';
GVL_test.stCase.aOuters[3].aPacks[2].nPackStatus := 5;
GVL_test.stCase.aOuters[3].aPacks[3].sPackCode   := 'PACK03OUTER3';
GVL_test.stCase.aOuters[3].aPacks[3].nPackStatus := 5;
GVL_test.stCase.aOuters[3].aPacks[4].sPackCode   := 'PACK04OUTER3';
GVL_test.stCase.aOuters[3].aPacks[4].nPackStatus := 5;
GVL_test.stCase.aOuters[3].aPacks[5].sPackCode   := 'PACK05OUTER3';
GVL_test.stCase.aOuters[3].aPacks[5].nPackStatus := 5;
GVL_test.stCase.aOuters[3].aPacks[6].sPackCode   := 'PACK06OUTER3';
GVL_test.stCase.aOuters[3].aPacks[6].nPackStatus := 5;
GVL_test.stCase.aOuters[3].aPacks[7].sPackCode   := 'PACK07OUTER3';
GVL_test.stCase.aOuters[3].aPacks[7].nPackStatus := 5;
GVL_test.stCase.aOuters[3].aPacks[8].sPackCode   := 'PACK08OUTER3';
GVL_test.stCase.aOuters[3].aPacks[8].nPackStatus := 5;
GVL_test.stCase.aOuters[3].aPacks[9].sPackCode   := 'PACK09OUTER3';
GVL_test.stCase.aOuters[3].aPacks[9].nPackStatus := 5;
GVL_test.stCase.aOuters[3].aPacks[10].sPackCode  := 'PACK10OUTER3';
GVL_test.stCase.aOuters[3].aPacks[10].nPackStatus := 5;

(* ===== OUTER 4 ===== *)
GVL_test.stCase.aOuters[4].sOuterCode    := 'OUTER4';
GVL_test.stCase.aOuters[4].nOutersStatus := 5;
// packs 1..10
GVL_test.stCase.aOuters[4].aPacks[1].sPackCode   := 'PACK01OUTER4';
GVL_test.stCase.aOuters[4].aPacks[1].nPackStatus := 5;
GVL_test.stCase.aOuters[4].aPacks[2].sPackCode   := 'PACK02OUTER4';
GVL_test.stCase.aOuters[4].aPacks[2].nPackStatus := 5;
GVL_test.stCase.aOuters[4].aPacks[3].sPackCode   := 'PACK03OUTER4';
GVL_test.stCase.aOuters[4].aPacks[3].nPackStatus := 5;
GVL_test.stCase.aOuters[4].aPacks[4].sPackCode   := 'PACK04OUTER4';
GVL_test.stCase.aOuters[4].aPacks[4].nPackStatus := 5;
GVL_test.stCase.aOuters[4].aPacks[5].sPackCode   := 'PACK05OUTER4';
GVL_test.stCase.aOuters[4].aPacks[5].nPackStatus := 5;
GVL_test.stCase.aOuters[4].aPacks[6].sPackCode   := 'PACK06OUTER4';
GVL_test.stCase.aOuters[4].aPacks[6].nPackStatus := 5;
GVL_test.stCase.aOuters[4].aPacks[7].sPackCode   := 'PACK07OUTER4';
GVL_test.stCase.aOuters[4].aPacks[7].nPackStatus := 5;
GVL_test.stCase.aOuters[4].aPacks[8].sPackCode   := 'PACK08OUTER4';
GVL_test.stCase.aOuters[4].aPacks[8].nPackStatus := 5;
GVL_test.stCase.aOuters[4].aPacks[9].sPackCode   := 'PACK09OUTER4';
GVL_test.stCase.aOuters[4].aPacks[9].nPackStatus := 5;
GVL_test.stCase.aOuters[4].aPacks[10].sPackCode  := 'PACK10OUTER4';
GVL_test.stCase.aOuters[4].aPacks[10].nPackStatus := 5;

(* ===== OUTER 5 ===== *)
GVL_test.stCase.aOuters[5].sOuterCode    := 'OUTER5';
GVL_test.stCase.aOuters[5].nOutersStatus := 5;
// packs 1..10
GVL_test.stCase.aOuters[5].aPacks[1].sPackCode   := 'PACK01OUTER5';
GVL_test.stCase.aOuters[5].aPacks[1].nPackStatus := 5;
GVL_test.stCase.aOuters[5].aPacks[2].sPackCode   := 'PACK02OUTER5';
GVL_test.stCase.aOuters[5].aPacks[2].nPackStatus := 5;
GVL_test.stCase.aOuters[5].aPacks[3].sPackCode   := 'PACK03OUTER5';
GVL_test.stCase.aOuters[5].aPacks[3].nPackStatus := 5;
GVL_test.stCase.aOuters[5].aPacks[4].sPackCode   := 'PACK04OUTER5';
GVL_test.stCase.aOuters[5].aPacks[4].nPackStatus := 5;
GVL_test.stCase.aOuters[5].aPacks[5].sPackCode   := 'PACK05OUTER5';
GVL_test.stCase.aOuters[5].aPacks[5].nPackStatus := 5;
GVL_test.stCase.aOuters[5].aPacks[6].sPackCode   := 'PACK06OUTER5';
GVL_test.stCase.aOuters[5].aPacks[6].nPackStatus := 5;
GVL_test.stCase.aOuters[5].aPacks[7].sPackCode   := 'PACK07OUTER5';
GVL_test.stCase.aOuters[5].aPacks[7].nPackStatus := 5;
GVL_test.stCase.aOuters[5].aPacks[8].sPackCode   := 'PACK08OUTER5';
GVL_test.stCase.aOuters[5].aPacks[8].nPackStatus := 5;
GVL_test.stCase.aOuters[5].aPacks[9].sPackCode   := 'PACK09OUTER5';
GVL_test.stCase.aOuters[5].aPacks[9].nPackStatus := 5;
GVL_test.stCase.aOuters[5].aPacks[10].sPackCode  := 'PACK10OUTER5';
GVL_test.stCase.aOuters[5].aPacks[10].nPackStatus := 5;

(* ===== OUTER 6 ===== *)
GVL_test.stCase.aOuters[6].sOuterCode    := 'OUTER6';
GVL_test.stCase.aOuters[6].nOutersStatus := 5;
// packs 1..10
GVL_test.stCase.aOuters[6].aPacks[1].sPackCode   := 'PACK01OUTER6';
GVL_test.stCase.aOuters[6].aPacks[1].nPackStatus := 5;
GVL_test.stCase.aOuters[6].aPacks[2].sPackCode   := 'PACK02OUTER6';
GVL_test.stCase.aOuters[6].aPacks[2].nPackStatus := 5;
GVL_test.stCase.aOuters[6].aPacks[3].sPackCode   := 'PACK03OUTER6';
GVL_test.stCase.aOuters[6].aPacks[3].nPackStatus := 5;
GVL_test.stCase.aOuters[6].aPacks[4].sPackCode   := 'PACK04OUTER6';
GVL_test.stCase.aOuters[6].aPacks[4].nPackStatus := 5;
GVL_test.stCase.aOuters[6].aPacks[5].sPackCode   := 'PACK05OUTER6';
GVL_test.stCase.aOuters[6].aPacks[5].nPackStatus := 5;
GVL_test.stCase.aOuters[6].aPacks[6].sPackCode   := 'PACK06OUTER6';
GVL_test.stCase.aOuters[6].aPacks[6].nPackStatus := 5;
GVL_test.stCase.aOuters[6].aPacks[7].sPackCode   := 'PACK07OUTER6';
GVL_test.stCase.aOuters[6].aPacks[7].nPackStatus := 5;
GVL_test.stCase.aOuters[6].aPacks[8].sPackCode   := 'PACK08OUTER6';
GVL_test.stCase.aOuters[6].aPacks[8].nPackStatus := 5;
GVL_test.stCase.aOuters[6].aPacks[9].sPackCode   := 'PACK09OUTER6';
GVL_test.stCase.aOuters[6].aPacks[9].nPackStatus := 5;
GVL_test.stCase.aOuters[6].aPacks[10].sPackCode  := 'PACK10OUTER6';
GVL_test.stCase.aOuters[6].aPacks[10].nPackStatus := 5;

(* ===== OUTER 7 ===== *)
GVL_test.stCase.aOuters[7].sOuterCode    := 'OUTER7';
GVL_test.stCase.aOuters[7].nOutersStatus := 5;
// packs 1..10
GVL_test.stCase.aOuters[7].aPacks[1].sPackCode   := 'PACK01OUTER7';
GVL_test.stCase.aOuters[7].aPacks[1].nPackStatus := 5;
GVL_test.stCase.aOuters[7].aPacks[2].sPackCode   := 'PACK02OUTER7';
GVL_test.stCase.aOuters[7].aPacks[2].nPackStatus := 5;
GVL_test.stCase.aOuters[7].aPacks[3].sPackCode   := 'PACK03OUTER7';
GVL_test.stCase.aOuters[7].aPacks[3].nPackStatus := 5;
GVL_test.stCase.aOuters[7].aPacks[4].sPackCode   := 'PACK04OUTER7';
GVL_test.stCase.aOuters[7].aPacks[4].nPackStatus := 5;
GVL_test.stCase.aOuters[7].aPacks[5].sPackCode   := 'PACK05OUTER7';
GVL_test.stCase.aOuters[7].aPacks[5].nPackStatus := 5;
GVL_test.stCase.aOuters[7].aPacks[6].sPackCode   := 'PACK06OUTER7';
GVL_test.stCase.aOuters[7].aPacks[6].nPackStatus := 5;
GVL_test.stCase.aOuters[7].aPacks[7].sPackCode   := 'PACK07OUTER7';
GVL_test.stCase.aOuters[7].aPacks[7].nPackStatus := 5;
GVL_test.stCase.aOuters[7].aPacks[8].sPackCode   := 'PACK08OUTER7';
GVL_test.stCase.aOuters[7].aPacks[8].nPackStatus := 5;
GVL_test.stCase.aOuters[7].aPacks[9].sPackCode   := 'PACK09OUTER7';
GVL_test.stCase.aOuters[7].aPacks[9].nPackStatus := 5;
GVL_test.stCase.aOuters[7].aPacks[10].sPackCode  := 'PACK10OUTER7';
GVL_test.stCase.aOuters[7].aPacks[10].nPackStatus := 5;

(* ===== OUTER 8 ===== *)
GVL_test.stCase.aOuters[8].sOuterCode    := 'OUTER8';
GVL_test.stCase.aOuters[8].nOutersStatus := 5;
// packs 1..10
GVL_test.stCase.aOuters[8].aPacks[1].sPackCode   := 'PACK01OUTER8';
GVL_test.stCase.aOuters[8].aPacks[1].nPackStatus := 5;
GVL_test.stCase.aOuters[8].aPacks[2].sPackCode   := 'PACK02OUTER8';
GVL_test.stCase.aOuters[8].aPacks[2].nPackStatus := 5;
GVL_test.stCase.aOuters[8].aPacks[3].sPackCode   := 'PACK03OUTER8';
GVL_test.stCase.aOuters[8].aPacks[3].nPackStatus := 5;
GVL_test.stCase.aOuters[8].aPacks[4].sPackCode   := 'PACK04OUTER8';
GVL_test.stCase.aOuters[8].aPacks[4].nPackStatus := 5;
GVL_test.stCase.aOuters[8].aPacks[5].sPackCode   := 'PACK05OUTER8';
GVL_test.stCase.aOuters[8].aPacks[5].nPackStatus := 5;
GVL_test.stCase.aOuters[8].aPacks[6].sPackCode   := 'PACK06OUTER8';
GVL_test.stCase.aOuters[8].aPacks[6].nPackStatus := 5;
GVL_test.stCase.aOuters[8].aPacks[7].sPackCode   := 'PACK07OUTER8';
GVL_test.stCase.aOuters[8].aPacks[7].nPackStatus := 5;
GVL_test.stCase.aOuters[8].aPacks[8].sPackCode   := 'PACK08OUTER8';
GVL_test.stCase.aOuters[8].aPacks[8].nPackStatus := 5;
GVL_test.stCase.aOuters[8].aPacks[9].sPackCode   := 'PACK09OUTER8';
GVL_test.stCase.aOuters[8].aPacks[9].nPackStatus := 5;
GVL_test.stCase.aOuters[8].aPacks[10].sPackCode  := 'PACK10OUTER8';
GVL_test.stCase.aOuters[8].aPacks[10].nPackStatus := 5;

(* ===== OUTER 9 ===== *)
GVL_test.stCase.aOuters[9].sOuterCode    := 'OUTER9';
GVL_test.stCase.aOuters[9].nOutersStatus := 5;
// packs 1..10
GVL_test.stCase.aOuters[9].aPacks[1].sPackCode   := 'PACK01OUTER9';
GVL_test.stCase.aOuters[9].aPacks[1].nPackStatus := 5;
GVL_test.stCase.aOuters[9].aPacks[2].sPackCode   := 'PACK02OUTER9';
GVL_test.stCase.aOuters[9].aPacks[2].nPackStatus := 5;
GVL_test.stCase.aOuters[9].aPacks[3].sPackCode   := 'PACK03OUTER9';
GVL_test.stCase.aOuters[9].aPacks[3].nPackStatus := 5;
GVL_test.stCase.aOuters[9].aPacks[4].sPackCode   := 'PACK04OUTER9';
GVL_test.stCase.aOuters[9].aPacks[4].nPackStatus := 5;
GVL_test.stCase.aOuters[9].aPacks[5].sPackCode   := 'PACK05OUTER9';
GVL_test.stCase.aOuters[9].aPacks[5].nPackStatus := 5;
GVL_test.stCase.aOuters[9].aPacks[6].sPackCode   := 'PACK06OUTER9';
GVL_test.stCase.aOuters[9].aPacks[6].nPackStatus := 5;
GVL_test.stCase.aOuters[9].aPacks[7].sPackCode   := 'PACK07OUTER9';
GVL_test.stCase.aOuters[9].aPacks[7].nPackStatus := 5;
GVL_test.stCase.aOuters[9].aPacks[8].sPackCode   := 'PACK08OUTER9';
GVL_test.stCase.aOuters[9].aPacks[8].nPackStatus := 5;
GVL_test.stCase.aOuters[9].aPacks[9].sPackCode   := 'PACK09OUTER9';
GVL_test.stCase.aOuters[9].aPacks[9].nPackStatus := 5;
GVL_test.stCase.aOuters[9].aPacks[10].sPackCode  := 'PACK10OUTER9';
GVL_test.stCase.aOuters[9].aPacks[10].nPackStatus := 5;

